LIN {X 0,Y 312.569,Z 218.829,A -85,B 0,C 180,E1 -15730.204,E2 -15730.204} C_VEL
LIN {X 0,Y 313.589,Z 221.679,A -85,B 0,C 180,E1 -15730.474,E2 -15730.474} C_VEL
LIN {X 0,Y 315.633,Z 224.126,A -85,B 0,C 180,E1 -15730.891,E2 -15730.891} C_VEL
LIN {X 0,Y 317.945,Z 227.629,A -85,B 0,C 180,E1 -15731.376,E2 -15731.376} C_VEL
LIN {X 0,Y 330.449,Z 246.954,A -85,B 0,C 180,E1 -15733.852,E2 -15733.852} C_VEL
LIN {X 0,Y 339.221,Z 262.018,A -85,B 0,C 180,E1 -15735.489,E2 -15735.489} C_VEL
LIN {X 0,Y 346.478,Z 276.506,A -85,B 0,C 180,E1 -15736.814,E2 -15736.814} C_VEL
LIN {X 0,Y 346.92,Z 277.621,A -85,B 0,C 180,E1 -15736.899,E2 -15736.899} C_VEL
LIN {X 0,Y 340.996,Z 419.211,A -85,B 0,C 180,E1 -15739.948,E2 -15739.948} C_VEL
LIN {X 0,Y 339.631,Z 436.329,A -85,B 0,C 180,E1 -15740.546,E2 -15740.546} C_VEL
LIN {X 0,Y 337.855,Z 452.225,A -85,B 0,C 180,E1 -15741.326,E2 -15741.326} C_VEL
LIN {X 0,Y 335.809,Z 467.786,A -85,B 0,C 180,E1 -15742.333,E2 -15742.333} C_VEL
LIN {X 0,Y 333.545,Z 482.265,A -85,B 0,C 180,E1 -15743.497,E2 -15743.497} C_VEL
LIN {X 0,Y 330.733,Z 497.251,A -85,B 0,C 180,E1 -15744.968,E2 -15744.968} C_VEL
LIN {X 0,Y 327.878,Z 510.986,A -85,B 0,C 180,E1 -15746.62,E2 -15746.62} C_VEL
LIN {X 0,Y 325.104,Z 523.666,A -85,B 0,C 180,E1 -15748.451,E2 -15748.451} C_VEL
LIN {X 0,Y 322.131,Z 536.293,A -85,B 0,C 180,E1 -15750.625,E2 -15750.625} C_VEL
LIN {X 0,Y 319.543,Z 547.053,A -85,B 0,C 180,E1 -15752.836,E2 -15752.836} C_VEL
LIN {X 0,Y 317.025,Z 557.47,A -85,B 0,C 180,E1 -15755.406,E2 -15755.406} C_VEL
LIN {X 0,Y 315.045,Z 566.149,A -85,B 0,C 180,E1 -15758.014,E2 -15758.014} C_VEL
LIN {X 0,Y 313.603,Z 572.562,A -85,B 0,C 180,E1 -15760.328,E2 -15760.328} C_VEL
LIN {X 0,Y 312.378,Z 578.726,A -85,B 0,C 180,E1 -15763.001,E2 -15763.001} C_VEL
LIN {X 0,Y 311.524,Z 583.601,A -85,B 0,C 180,E1 -15765.707,E2 -15765.707} C_VEL
LIN {X 0,Y 310.896,Z 587.382,A -85,B 0,C 180,E1 -15768.449,E2 -15768.449} C_VEL
LIN {X 0,Y 310.55,Z 590.089,A -85,B 0,C 180,E1 -15771.228,E2 -15771.228} C_VEL
LIN {X 0,Y 310.352,Z 591.614,A -85,B 0,C 180,E1 -15774.054,E2 -15774.054} C_VEL
LIN {X 0,Y 310.334,Z 592.053,A -85,B 0,C 180,E1 -15776.931,E2 -15776.931} C_VEL
LIN {X 0,Y 310.51,Z 591.326,A -85,B 0,C 180,E1 -15779.863,E2 -15779.863} C_VEL
LIN {X 0,Y 310.927,Z 588.932,A -85,B 0,C 180,E1 -15783.246,E2 -15783.246} C_VEL
LIN {X 0,Y 311.753,Z 584.791,A -85,B 0,C 180,E1 -15786.683,E2 -15786.683} C_VEL
LIN {X 0,Y 312.79,Z 579.753,A -85,B 0,C 180,E1 -15789.629,E2 -15789.629} C_VEL
LIN {X 0,Y 314.219,Z 573.616,A -85,B 0,C 180,E1 -15792.431,E2 -15792.431} C_VEL
LIN {X 0,Y 315.326,Z 569.216,A -85,B 0,C 180,E1 -15794.117,E2 -15794.117} C_VEL
LIN {X 0,Y 315.393,Z 566.63,A -85,B 0,C 180,E1 -15795.081,E2 -15795.081} C_VEL
LIN {X 0,Y 312.533,Z 557.734,A -85,B 0,C 180,E1 -15798.272,E2 -15798.272} C_VEL
LIN {X 0,Y 312.862,Z 554.516,A -85,B 0,C 180,E1 -15799.184,E2 -15799.184} C_VEL
LIN {X 0,Y 315.976,Z 543.99,A -85,B 0,C 180,E1 -15801.682,E2 -15801.682} C_VEL
LIN {X 0,Y 319.14,Z 533.152,A -85,B 0,C 180,E1 -15803.831,E2 -15803.831} C_VEL
LIN {X 0,Y 322.204,Z 521.844,A -85,B 0,C 180,E1 -15805.734,E2 -15805.734} C_VEL
LIN {X 0,Y 325.653,Z 508.462,A -85,B 0,C 180,E1 -15807.602,E2 -15807.602} C_VEL
LIN {X 0,Y 328.772,Z 495.26,A -85,B 0,C 180,E1 -15809.134,E2 -15809.134} C_VEL
LIN {X 0,Y 331.674,Z 481.349,A -85,B 0,C 180,E1 -15810.484,E2 -15810.484} C_VEL
LIN {X 0,Y 334.505,Z 465.783,A -85,B 0,C 180,E1 -15811.703,E2 -15811.703} C_VEL
LIN {X 0,Y 336.821,Z 449.961,A -85,B 0,C 180,E1 -15812.675,E2 -15812.675} C_VEL
LIN {X 0,Y 338.694,Z 433.873,A -85,B 0,C 180,E1 -15813.419,E2 -15813.419} C_VEL
LIN {X 0,Y 340.182,Z 416.337,A -85,B 0,C 180,E1 -15813.973,E2 -15813.973} C_VEL
LIN {X 0,Y 346.65,Z 282.972,A -85,B 0,C 180,E1 -15816.935,E2 -15816.935} C_VEL
LIN {X 0,Y 340.142,Z 270.114,A -85,B 0,C 180,E1 -15818.442,E2 -15818.442} C_VEL
LIN {X 0,Y 335.198,Z 261.466,A -85,B 0,C 180,E1 -15819.629,E2 -15819.629} C_VEL
LIN {X 0,Y 328.703,Z 251.5,A -85,B 0,C 180,E1 -15821.263,E2 -15821.263} C_VEL
LIN {X 0,Y 322.882,Z 243.203,A -85,B 0,C 180,E1 -15822.83,E2 -15822.83} C_VEL
LIN {X 0,Y 319.655,Z 238.87,A -85,B 0,C 180,E1 -15823.746,E2 -15823.746} C_VEL
LIN {X 0,Y 316.6,Z 234.714,A -85,B 0,C 180,E1 -15824.664,E2 -15824.664} C_VEL
LIN {X 0,Y 313.996,Z 231.244,A -85,B 0,C 180,E1 -15825.477,E2 -15825.477} C_VEL
LIN {X 0,Y 313.147,Z 230.084,A -85,B 0,C 180,E1 -15825.753,E2 -15825.753} C_VEL
LIN {X 0,Y 310.657,Z 227.254,A -85,B 0,C 180,E1 -15826.559,E2 -15826.559} C_VEL
LIN {X 0,Y 309.552,Z 225.243,A -85,B 0,C 180,E1 -15826.961,E2 -15826.961} C_VEL
LIN {X 0,Y 307.098,Z 223.278,A -85,B 0,C 180,E1 -15827.779,E2 -15827.779} C_VEL
LIN {X 0,Y 305.86,Z 220.899,A -85,B 0,C 180,E1 -15828.275,E2 -15828.275} C_VEL
LIN {X 0,Y 305.62,Z 219.711,A -85,B 0,C 180,E1 -15828.434,E2 -15828.434} C_VEL
LIN {X 0,Y 305.766,Z 219.711,A -85,B 0,C 180,E1 -15832.073,E2 -15832.073} C_VEL
LIN {X 0,Y 305.676,Z 219.722,A -85,B 0,C 180,E1 -15834.723,E2 -15834.723} C_VEL
LIN {X 0,Y 305.951,Z 219.685,A -85,B 0,C 180,E1 -15838.684,E2 -15838.684} C_VEL
LIN {X 0,Y 305.951,Z 219.686,A -85,B 0,C 180,E1 -15841.316,E2 -15841.316} C_VEL
LIN {X 0,Y 305.837,Z 219.7,A -85,B 0,C 180,E1 -15846.598,E2 -15846.598} C_VEL
LIN {X 0,Y 305.698,Z 219.717,A -85,B 0,C 180,E1 -15849.261,E2 -15849.261} C_VEL
LIN {X 0,Y 305.583,Z 219.729,A -85,B 0,C 180,E1 -15853.296,E2 -15853.296} C_VEL
LIN {X 0,Y 305.588,Z 219.727,A -85,B 0,C 180,E1 -15856.02,E2 -15856.02} C_VEL
LIN {X 0,Y 305.571,Z 219.729,A -85,B 0,C 180,E1 -15859.445,E2 -15859.445} C_VEL
LIN {X 0,Y 305.486,Z 219.746,A -85,B 0,C 180,E1 -15863.042,E2 -15863.042} C_VEL
LIN {X 0,Y 305.526,Z 219.736,A -85,B 0,C 180,E1 -15866.221,E2 -15866.221} C_VEL
LIN {X 0,Y 305.483,Z 219.742,A -85,B 0,C 180,E1 -15869.047,E2 -15869.047} C_VEL
LIN {X 0,Y 305.437,Z 219.751,A -85,B 0,C 180,E1 -15871.953,E2 -15871.953} C_VEL
LIN {X 0,Y 305.514,Z 219.86,A -85,B 0,C 180,E1 -15876.018,E2 -15876.018} C_VEL
LIN {X 0,Y 305.951,Z 221.601,A -85,B 0,C 180,E1 -15876.673,E2 -15876.673} C_VEL
LIN {X 0,Y 307.613,Z 224.865,A -85,B 0,C 180,E1 -15878.087,E2 -15878.087} C_VEL
LIN {X 0,Y 314.06,Z 233.766,A -85,B 0,C 180,E1 -15880.282,E2 -15880.282} C_VEL
LIN {X 0,Y 317.349,Z 238.402,A -85,B 0,C 180,E1 -15881.308,E2 -15881.308} C_VEL
LIN {X 0,Y 323.89,Z 248.152,A -85,B 0,C 180,E1 -15883.218,E2 -15883.218} C_VEL
LIN {X 0,Y 330.61,Z 259.152,A -85,B 0,C 180,E1 -15885.03,E2 -15885.03} C_VEL
LIN {X 0,Y 337.16,Z 270.828,A -85,B 0,C 180,E1 -15886.682,E2 -15886.682} C_VEL
LIN {X 0,Y 344.759,Z 286.276,A -85,B 0,C 180,E1 -15888.492,E2 -15888.492} C_VEL
LIN {X 0,Y 346.397,Z 289.941,A -85,B 0,C 180,E1 -15888.87,E2 -15888.87} C_VEL
LIN {X 0,Y 342.866,Z 363.369,A -85,B 0,C 180,E1 -15890.493,E2 -15890.493} C_VEL
LIN {X 0,Y 339.405,Z 435.134,A -85,B 0,C 180,E1 -15892.117,E2 -15892.117} C_VEL
LIN {X 0,Y 337.581,Z 452.624,A -85,B 0,C 180,E1 -15892.709,E2 -15892.709} C_VEL
LIN {X 0,Y 335.323,Z 469.014,A -85,B 0,C 180,E1 -15893.509,E2 -15893.509} C_VEL
LIN {X 0,Y 332.78,Z 484.339,A -85,B 0,C 180,E1 -15894.496,E2 -15894.496} C_VEL
LIN {X 0,Y 329.551,Z 500.237,A -85,B 0,C 180,E1 -15895.774,E2 -15895.774} C_VEL
LIN {X 0,Y 326.409,Z 514.583,A -85,B 0,C 180,E1 -15897.22,E2 -15897.22} C_VEL
LIN {X 0,Y 323.002,Z 528.277,A -85,B 0,C 180,E1 -15898.886,E2 -15898.886} C_VEL
LIN {X 0,Y 319.679,Z 540.731,A -85,B 0,C 180,E1 -15900.716,E2 -15900.716} C_VEL
LIN {X 0,Y 316.341,Z 552.857,A -85,B 0,C 180,E1 -15902.839,E2 -15902.839} C_VEL
LIN {X 0,Y 313.259,Z 563.818,A -85,B 0,C 180,E1 -15905.125,E2 -15905.125} C_VEL
LIN {X 0,Y 310.401,Z 574.161,A -85,B 0,C 180,E1 -15907.714,E2 -15907.714} C_VEL
LIN {X 0,Y 308.171,Z 582.797,A -85,B 0,C 180,E1 -15910.344,E2 -15910.344} C_VEL
LIN {X 0,Y 306.182,Z 590.845,A -85,B 0,C 180,E1 -15913.327,E2 -15913.327} C_VEL
LIN {X 0,Y 304.989,Z 596.69,A -85,B 0,C 180,E1 -15915.999,E2 -15915.999} C_VEL
LIN {X 0,Y 304.163,Z 601.391,A -85,B 0,C 180,E1 -15918.674,E2 -15918.674} C_VEL
LIN {X 0,Y 303.817,Z 604.222,A -85,B 0,C 180,E1 -15920.682,E2 -15920.682} C_VEL
LIN {X 0,Y 303.618,Z 607.009,A -85,B 0,C 180,E1 -15923.354,E2 -15923.354} C_VEL
LIN {X 0,Y 303.566,Z 608.885,A -85,B 0,C 180,E1 -15926.018,E2 -15926.018} C_VEL
LIN {X 0,Y 303.575,Z 609.682,A -85,B 0,C 180,E1 -15928.674,E2 -15928.674} C_VEL
LIN {X 0,Y 303.575,Z 609.59,A -85,B 0,C 180,E1 -15931.327,E2 -15931.327} C_VEL
LIN {X 0,Y 303.599,Z 608.416,A -85,B 0,C 180,E1 -15933.983,E2 -15933.983} C_VEL
LIN {X 0,Y 303.618,Z 606.325,A -85,B 0,C 180,E1 -15936.646,E2 -15936.646} C_VEL
LIN {X 0,Y 303.808,Z 603.111,A -85,B 0,C 180,E1 -15939.319,E2 -15939.319} C_VEL
LIN {X 0,Y 304.305,Z 598.874,A -85,B 0,C 180,E1 -15941.997,E2 -15941.997} C_VEL
LIN {X 0,Y 305.262,Z 593.244,A -85,B 0,C 180,E1 -15944.77,E2 -15944.77} C_VEL
LIN {X 0,Y 306.403,Z 586.766,A -85,B 0,C 180,E1 -15947.349,E2 -15947.349} C_VEL
LIN {X 0,Y 308.156,Z 578.729,A -85,B 0,C 180,E1 -15950.005,E2 -15950.005} C_VEL
LIN {X 0,Y 310.396,Z 569.109,A -85,B 0,C 180,E1 -15952.639,E2 -15952.639} C_VEL
LIN {X 0,Y 313.287,Z 557.586,A -85,B 0,C 180,E1 -15955.229,E2 -15955.229} C_VEL
LIN {X 0,Y 315.771,Z 547.009,A -85,B 0,C 180,E1 -15957.22,E2 -15957.22} C_VEL
LIN {X 0,Y 318.71,Z 534.598,A -85,B 0,C 180,E1 -15959.202,E2 -15959.202} C_VEL
LIN {X 0,Y 321.65,Z 521.958,A -85,B 0,C 180,E1 -15960.895,E2 -15960.895} C_VEL
LIN {X 0,Y 324.777,Z 507.198,A -85,B 0,C 180,E1 -15962.525,E2 -15962.525} C_VEL
LIN {X 0,Y 327.701,Z 491.892,A -85,B 0,C 180,E1 -15963.89,E2 -15963.89} C_VEL
LIN {X 0,Y 330.138,Z 476.607,A -85,B 0,C 180,E1 -15964.991,E2 -15964.991} C_VEL
LIN {X 0,Y 332.302,Z 459.741,A -85,B 0,C 180,E1 -15965.937,E2 -15965.937} C_VEL
LIN {X 0,Y 334.07,Z 443.602,A -85,B 0,C 180,E1 -15966.582,E2 -15966.582} C_VEL
LIN {X 0,Y 335.225,Z 427.63,A -85,B 0,C 180,E1 -15967.018,E2 -15967.018} C_VEL
LIN {X 0,Y 340.97,Z 287.709,A -85,B 0,C 180,E1 -15970.075,E2 -15970.075} C_VEL
LIN {X 0,Y 333.834,Z 272.618,A -85,B 0,C 180,E1 -15971.436,E2 -15971.436} C_VEL
LIN {X 0,Y 324.567,Z 254.726,A -85,B 0,C 180,E1 -15973.279,E2 -15973.279} C_VEL
LIN {X 0,Y 314.082,Z 236.733,A -85,B 0,C 180,E1 -15975.47,E2 -15975.47} C_VEL
LIN {X 0,Y 308.14,Z 226.968,A -85,B 0,C 180,E1 -15976.825,E2 -15976.825} C_VEL
LIN {X 0,Y 305.419,Z 219.741,A -85,B 0,C 180,E1 -15978.827,E2 -15978.827} C_VEL
LIN {X 0,Y 305.46,Z 219.751,A -85,B 0,C 180,E1 -15981.595,E2 -15981.595} C_VEL
LIN {X 0,Y 305.46,Z 219.738,A -85,B 0,C 180,E1 -15984.887,E2 -15984.887} C_VEL
LIN {X 0,Y 305.447,Z 219.727,A -85,B 0,C 180,E1 -15988.356,E2 -15988.356} C_VEL
LIN {X 0,Y 305.512,Z 219.744,A -85,B 0,C 180,E1 -15991.113,E2 -15991.113} C_VEL
LIN {X 0,Y 305.563,Z 219.708,A -85,B 0,C 180,E1 -15994.087,E2 -15994.087} C_VEL
LIN {X 0,Y 305.493,Z 219.737,A -85,B 0,C 180,E1 -15998.402,E2 -15998.402} C_VEL
LIN {X 0,Y 305.541,Z 219.706,A -85,B 0,C 180,E1 -16001.215,E2 -16001.215} C_VEL
LIN {X 0,Y 305.624,Z 219.724,A -85,B 0,C 180,E1 -16005.348,E2 -16005.348} C_VEL
LIN {X 0,Y 305.622,Z 219.693,A -85,B 0,C 180,E1 -16009.399,E2 -16009.399} C_VEL
LIN {X 0,Y 305.769,Z 219.708,A -85,B 0,C 180,E1 -16012.073,E2 -16012.073} C_VEL
LIN {X 0,Y 305.679,Z 219.702,A -85,B 0,C 180,E1 -16014.723,E2 -16014.723} C_VEL
LIN {X 0,Y 305.953,Z 219.652,A -85,B 0,C 180,E1 -16018.684,E2 -16018.684} C_VEL
LIN {X 0,Y 305.955,Z 219.685,A -85,B 0,C 180,E1 -16021.316,E2 -16021.316} C_VEL
LIN {X 0,Y 305.84,Z 219.686,A -85,B 0,C 180,E1 -16026.601,E2 -16026.601} C_VEL
LIN {X 0,Y 305.702,Z 219.715,A -85,B 0,C 180,E1 -16029.261,E2 -16029.261} C_VEL
LIN {X 0,Y 305.586,Z 219.717,A -85,B 0,C 180,E1 -16033.296,E2 -16033.296} C_VEL
LIN {X 0,Y 305.592,Z 219.728,A -85,B 0,C 180,E1 -16036.02,E2 -16036.02} C_VEL
LIN {X 0,Y 305.575,Z 219.709,A -85,B 0,C 180,E1 -16039.445,E2 -16039.445} C_VEL
LIN {X 0,Y 305.489,Z 219.742,A -85,B 0,C 180,E1 -16043.041,E2 -16043.041} C_VEL
LIN {X 0,Y 305.553,Z 219.715,A -85,B 0,C 180,E1 -16046.23,E2 -16046.23} C_VEL
LIN {X 0,Y 305.502,Z 219.743,A -85,B 0,C 180,E1 -16049.052,E2 -16049.052} C_VEL
LIN {X 0,Y 305.464,Z 219.736,A -85,B 0,C 180,E1 -16053.517,E2 -16053.517} C_VEL
LIN {X 0,Y 305.471,Z 219.738,A -85,B 0,C 180,E1 -16056.74,E2 -16056.74} C_VEL
LIN {X 0,Y 305.454,Z 219.748,A -85,B 0,C 180,E1 -16060.6,E2 -16060.6} C_VEL
LIN {X 0,Y 305.424,Z 219.735,A -85,B 0,C 180,E1 -16063.655,E2 -16063.655} C_VEL
LIN {X 0,Y 305.454,Z 219.744,A -85,B 0,C 180,E1 -16067.414,E2 -16067.414} C_VEL
LIN {X 0,Y 305.475,Z 219.747,A -85,B 0,C 180,E1 -16071.598,E2 -16071.598} C_VEL
LIN {X 0,Y 305.461,Z 219.736,A -85,B 0,C 180,E1 -16074.887,E2 -16074.887} C_VEL
LIN {X 0,Y 305.451,Z 219.735,A -85,B 0,C 180,E1 -16078.355,E2 -16078.355} C_VEL
LIN {X 0,Y 305.52,Z 219.742,A -85,B 0,C 180,E1 -16081.114,E2 -16081.114} C_VEL
LIN {X 0,Y 305.571,Z 219.732,A -85,B 0,C 180,E1 -16084.088,E2 -16084.088} C_VEL
LIN {X 0,Y 305.511,Z 219.733,A -85,B 0,C 180,E1 -16088.722,E2 -16088.722} C_VEL
LIN {X 0,Y 305.526,Z 219.862,A -85,B 0,C 180,E1 -16089.021,E2 -16089.021} C_VEL
LIN {X 0,Y 306.552,Z 222.628,A -85,B 0,C 180,E1 -16089.295,E2 -16089.295} C_VEL
LIN {X 0,Y 308.681,Z 225.163,A -85,B 0,C 180,E1 -16089.75,E2 -16089.75} C_VEL
LIN {X 0,Y 310.838,Z 228.393,A -85,B 0,C 180,E1 -16090.225,E2 -16090.225} C_VEL
LIN {X 0,Y 321.959,Z 245.231,A -85,B 0,C 180,E1 -16092.545,E2 -16092.545} C_VEL
LIN {X 0,Y 330.594,Z 259.454,A -85,B 0,C 180,E1 -16094.234,E2 -16094.234} C_VEL
LIN {X 0,Y 336.365,Z 269.967,A -85,B 0,C 180,E1 -16095.329,E2 -16095.329} C_VEL
LIN {X 0,Y 341.118,Z 279.595,A -85,B 0,C 180,E1 -16096.219,E2 -16096.219} C_VEL
LIN {X 0,Y 335.132,Z 419.139,A -85,B 0,C 180,E1 -16099.274,E2 -16099.274} C_VEL
LIN {X 0,Y 333.716,Z 436.368,A -85,B 0,C 180,E1 -16099.879,E2 -16099.879} C_VEL
LIN {X 0,Y 331.815,Z 452.948,A -85,B 0,C 180,E1 -16100.706,E2 -16100.706} C_VEL
LIN {X 0,Y 329.677,Z 468.427,A -85,B 0,C 180,E1 -16101.726,E2 -16101.726} C_VEL
LIN {X 0,Y 327.361,Z 482.815,A -85,B 0,C 180,E1 -16102.909,E2 -16102.909} C_VEL
LIN {X 0,Y 324.448,Z 497.796,A -85,B 0,C 180,E1 -16104.405,E2 -16104.405} C_VEL
LIN {X 0,Y 321.504,Z 511.467,A -85,B 0,C 180,E1 -16106.083,E2 -16106.083} C_VEL
LIN {X 0,Y 318.822,Z 523.141,A -85,B 0,C 180,E1 -16107.789,E2 -16107.789} C_VEL
LIN {X 0,Y 315.998,Z 534.828,A -85,B 0,C 180,E1 -16109.795,E2 -16109.795} C_VEL
LIN {X 0,Y 313.384,Z 545.28,A -85,B 0,C 180,E1 -16111.927,E2 -16111.927} C_VEL
LIN {X 0,Y 310.805,Z 555.383,A -85,B 0,C 180,E1 -16114.383,E2 -16114.383} C_VEL
LIN {X 0,Y 308.713,Z 563.923,A -85,B 0,C 180,E1 -16116.864,E2 -16116.864} C_VEL
LIN {X 0,Y 307.114,Z 570.736,A -85,B 0,C 180,E1 -16119.217,E2 -16119.217} C_VEL
LIN {X 0,Y 305.74,Z 577.196,A -85,B 0,C 180,E1 -16121.939,E2 -16121.939} C_VEL
LIN {X 0,Y 304.708,Z 582.483,A -85,B 0,C 180,E1 -16124.697,E2 -16124.697} C_VEL
LIN {X 0,Y 303.991,Z 586.603,A -85,B 0,C 180,E1 -16127.49,E2 -16127.49} C_VEL
LIN {X 0,Y 303.515,Z 589.576,A -85,B 0,C 180,E1 -16130.323,E2 -16130.323} C_VEL
LIN {X 0,Y 303.271,Z 591.502,A -85,B 0,C 180,E1 -16133.2,E2 -16133.2} C_VEL
LIN {X 0,Y 303.219,Z 592.26,A -85,B 0,C 180,E1 -16136.127,E2 -16136.127} C_VEL
LIN {X 0,Y 303.36,Z 591.84,A -85,B 0,C 180,E1 -16139.111,E2 -16139.111} C_VEL
LIN {X 0,Y 303.642,Z 590.209,A -85,B 0,C 180,E1 -16142.163,E2 -16142.163} C_VEL
LIN {X 0,Y 304.273,Z 587.239,A -85,B 0,C 180,E1 -16145.27,E2 -16145.27} C_VEL
LIN {X 0,Y 305.238,Z 582.667,A -85,B 0,C 180,E1 -16148.479,E2 -16148.479} C_VEL
LIN {X 0,Y 306.689,Z 576.602,A -85,B 0,C 180,E1 -16151.647,E2 -16151.647} C_VEL
LIN {X 0,Y 308.505,Z 569.741,A -85,B 0,C 180,E1 -16154.467,E2 -16154.467} C_VEL
LIN {X 0,Y 310.901,Z 561.24,A -85,B 0,C 180,E1 -16157.3,E2 -16157.3} C_VEL
LIN {X 0,Y 312.862,Z 554.516,A -85,B 0,C 180,E1 -16159.184,E2 -16159.184} C_VEL
LIN {X 0,Y 313.25,Z 551.252,A -85,B 0,C 180,E1 -16160.082,E2 -16160.082} C_VEL
LIN {X 0,Y 311.457,Z 540.284,A -85,B 0,C 180,E1 -16163.088,E2 -16163.088} C_VEL
LIN {X 0,Y 312.049,Z 536.454,A -85,B 0,C 180,E1 -16163.913,E2 -16163.913} C_VEL
LIN {X 0,Y 315.472,Z 524.42,A -85,B 0,C 180,E1 -16166.05,E2 -16166.05} C_VEL
LIN {X 0,Y 319.091,Z 511.357,A -85,B 0,C 180,E1 -16167.966,E2 -16167.966} C_VEL
LIN {X 0,Y 322.175,Z 498.973,A -85,B 0,C 180,E1 -16169.502,E2 -16169.502} C_VEL
LIN {X 0,Y 325.456,Z 484.325,A -85,B 0,C 180,E1 -16170.992,E2 -16170.992} C_VEL
LIN {X 0,Y 328.363,Z 469.451,A -85,B 0,C 180,E1 -16172.218,E2 -16172.218} C_VEL
LIN {X 0,Y 330.743,Z 454.966,A -85,B 0,C 180,E1 -16173.182,E2 -16173.182} C_VEL
LIN {X 0,Y 332.751,Z 439.646,A -85,B 0,C 180,E1 -16173.983,E2 -16173.983} C_VEL
LIN {X 0,Y 334.379,Z 423.357,A -85,B 0,C 180,E1 -16174.582,E2 -16174.582} C_VEL
LIN {X 0,Y 335.785,Z 398.674,A -85,B 0,C 180,E1 -16175.187,E2 -16175.187} C_VEL
LIN {X 0,Y 341.519,Z 285.669,A -85,B 0,C 180,E1 -16177.71,E2 -16177.71} C_VEL
LIN {X 0,Y 335.762,Z 274.293,A -85,B 0,C 180,E1 -16179.098,E2 -16179.098} C_VEL
LIN {X 0,Y 331.39,Z 266.453,A -85,B 0,C 180,E1 -16180.198,E2 -16180.198} C_VEL
LIN {X 0,Y 324.525,Z 255.848,A -85,B 0,C 180,E1 -16181.992,E2 -16181.992} C_VEL
LIN {X 0,Y 319.039,Z 248.008,A -85,B 0,C 180,E1 -16183.535,E2 -16183.535} C_VEL
LIN {X 0,Y 316.21,Z 244.147,A -85,B 0,C 180,E1 -16184.377,E2 -16184.377} C_VEL
LIN {X 0,Y 313.482,Z 240.367,A -85,B 0,C 180,E1 -16185.228,E2 -16185.228} C_VEL
LIN {X 0,Y 310.182,Z 235.952,A -85,B 0,C 180,E1 -16186.307,E2 -16186.307} C_VEL
LIN {X 0,Y 307.54,Z 232.58,A -85,B 0,C 180,E1 -16187.21,E2 -16187.21} C_VEL
LIN {X 0,Y 306.712,Z 231.384,A -85,B 0,C 180,E1 -16187.511,E2 -16187.511} C_VEL
LIN {X 0,Y 304.265,Z 228.977,A -85,B 0,C 180,E1 -16188.382,E2 -16188.382} C_VEL
LIN {X 0,Y 302.648,Z 226.153,A -85,B 0,C 180,E1 -16189.04,E2 -16189.04} C_VEL
LIN {X 0,Y 300.243,Z 224.347,A -85,B 0,C 180,E1 -16189.932,E2 -16189.932} C_VEL
LIN {X 0,Y 298.977,Z 222.103,A -85,B 0,C 180,E1 -16190.486,E2 -16190.486} C_VEL
LIN {X 0,Y 298.669,Z 220.592,A -85,B 0,C 180,E1 -16190.729,E2 -16190.729} C_VEL
LIN {X 0,Y 298.769,Z 220.577,A -85,B 0,C 180,E1 -16193.245,E2 -16193.245} C_VEL
LIN {X 0,Y 298.918,Z 220.56,A -85,B 0,C 180,E1 -16198.653,E2 -16198.653} C_VEL
LIN {X 0,Y 298.918,Z 220.562,A -85,B 0,C 180,E1 -16201.347,E2 -16201.347} C_VEL
LIN {X 0,Y 298.782,Z 220.58,A -85,B 0,C 180,E1 -16206.754,E2 -16206.754} C_VEL
LIN {X 0,Y 298.63,Z 220.599,A -85,B 0,C 180,E1 -16209.482,E2 -16209.482} C_VEL
LIN {X 0,Y 298.547,Z 220.604,A -85,B 0,C 180,E1 -16213.616,E2 -16213.616} C_VEL
LIN {X 0,Y 298.543,Z 220.604,A -85,B 0,C 180,E1 -16216.409,E2 -16216.409} C_VEL
LIN {X 0,Y 298.506,Z 220.61,A -85,B 0,C 180,E1 -16219.655,E2 -16219.655} C_VEL
LIN {X 0,Y 298.453,Z 220.618,A -85,B 0,C 180,E1 -16223.598,E2 -16223.598} C_VEL
LIN {X 0,Y 298.482,Z 220.613,A -85,B 0,C 180,E1 -16226.575,E2 -16226.575} C_VEL
LIN {X 0,Y 298.411,Z 220.624,A -85,B 0,C 180,E1 -16229.642,E2 -16229.642} C_VEL
LIN {X 0,Y 298.426,Z 220.685,A -85,B 0,C 180,E1 -16233.907,E2 -16233.907} C_VEL
LIN {X 0,Y 299.354,Z 223.361,A -85,B 0,C 180,E1 -16235.112,E2 -16235.112} C_VEL
LIN {X 0,Y 300.441,Z 224.75,A -85,B 0,C 180,E1 -16235.789,E2 -16235.789} C_VEL
LIN {X 0,Y 302.599,Z 228.072,A -85,B 0,C 180,E1 -16236.674,E2 -16236.674} C_VEL
LIN {X 0,Y 305.308,Z 231.386,A -85,B 0,C 180,E1 -16237.694,E2 -16237.694} C_VEL
LIN {X 0,Y 311.192,Z 239.615,A -85,B 0,C 180,E1 -16239.766,E2 -16239.766} C_VEL
LIN {X 0,Y 314.353,Z 244.238,A -85,B 0,C 180,E1 -16240.795,E2 -16240.795} C_VEL
LIN {X 0,Y 320.383,Z 253.329,A -85,B 0,C 180,E1 -16242.62,E2 -16242.62} C_VEL
LIN {X 0,Y 327.747,Z 265.663,A -85,B 0,C 180,E1 -16244.677,E2 -16244.677} C_VEL
LIN {X 0,Y 333.797,Z 276.856,A -85,B 0,C 180,E1 -16246.256,E2 -16246.256} C_VEL
LIN {X 0,Y 340.947,Z 291.732,A -85,B 0,C 180,E1 -16248.018,E2 -16248.018} C_VEL
LIN {X 0,Y 341.275,Z 292.503,A -85,B 0,C 180,E1 -16248.099,E2 -16248.099} C_VEL
LIN {X 0,Y 335.393,Z 408.882,A -85,B 0,C 180,E1 -16250.69,E2 -16250.69} C_VEL
LIN {X 0,Y 333.935,Z 436.305,A -85,B 0,C 180,E1 -16251.357,E2 -16251.357} C_VEL
LIN {X 0,Y 332.089,Z 453.273,A -85,B 0,C 180,E1 -16251.948,E2 -16251.948} C_VEL
LIN {X 0,Y 329.69,Z 469.884,A -85,B 0,C 180,E1 -16252.782,E2 -16252.782} C_VEL
LIN {X 0,Y 327.044,Z 484.917,A -85,B 0,C 180,E1 -16253.776,E2 -16253.776} C_VEL
LIN {X 0,Y 323.728,Z 500.616,A -85,B 0,C 180,E1 -16255.07,E2 -16255.07} C_VEL
LIN {X 0,Y 320.429,Z 514.814,A -85,B 0,C 180,E1 -16256.523,E2 -16256.523} C_VEL
LIN {X 0,Y 316.9,Z 528.499,A -85,B 0,C 180,E1 -16258.217,E2 -16258.217} C_VEL
LIN {X 0,Y 313.457,Z 540.884,A -85,B 0,C 180,E1 -16260.076,E2 -16260.076} C_VEL
LIN {X 0,Y 310.184,Z 552.186,A -85,B 0,C 180,E1 -16262.084,E2 -16262.084} C_VEL
LIN {X 0,Y 307.16,Z 562.462,A -85,B 0,C 180,E1 -16264.233,E2 -16264.233} C_VEL
LIN {X 0,Y 304.089,Z 572.922,A -85,B 0,C 180,E1 -16266.866,E2 -16266.866} C_VEL
LIN {X 0,Y 301.634,Z 581.728,A -85,B 0,C 180,E1 -16269.544,E2 -16269.544} C_VEL
LIN {X 0,Y 299.67,Z 589.128,A -85,B 0,C 180,E1 -16272.25,E2 -16272.25} C_VEL
LIN {X 0,Y 298.232,Z 595.426,A -85,B 0,C 180,E1 -16275.057,E2 -16275.057} C_VEL
LIN {X 0,Y 297.327,Z 600.166,A -85,B 0,C 180,E1 -16277.718,E2 -16277.718} C_VEL
LIN {X 0,Y 296.736,Z 604.069,A -85,B 0,C 180,E1 -16280.457,E2 -16280.457} C_VEL
LIN {X 0,Y 296.533,Z 606.841,A -85,B 0,C 180,E1 -16283.195,E2 -16283.195} C_VEL
LIN {X 0,Y 296.468,Z 608.698,A -85,B 0,C 180,E1 -16285.922,E2 -16285.922} C_VEL
LIN {X 0,Y 296.493,Z 609.482,A -85,B 0,C 180,E1 -16288.642,E2 -16288.642} C_VEL
LIN {X 0,Y 296.494,Z 609.369,A -85,B 0,C 180,E1 -16291.359,E2 -16291.359} C_VEL
LIN {X 0,Y 296.496,Z 608.18,A -85,B 0,C 180,E1 -16294.078,E2 -16294.078} C_VEL
LIN {X 0,Y 296.533,Z 606.063,A -85,B 0,C 180,E1 -16296.806,E2 -16296.806} C_VEL
LIN {X 0,Y 296.821,Z 601.913,A -85,B 0,C 180,E1 -16300.229,E2 -16300.229} C_VEL
LIN {X 0,Y 297.726,Z 596.03,A -85,B 0,C 180,E1 -16303.654,E2 -16303.654} C_VEL
LIN {X 0,Y 298.784,Z 589.928,A -85,B 0,C 180,E1 -16306.396,E2 -16306.396} C_VEL
LIN {X 0,Y 300.449,Z 582.559,A -85,B 0,C 180,E1 -16309.116,E2 -16309.116} C_VEL
LIN {X 0,Y 302.462,Z 573.722,A -85,B 0,C 180,E1 -16311.825,E2 -16311.825} C_VEL
LIN {X 0,Y 305.175,Z 563.162,A -85,B 0,C 180,E1 -16314.49,E2 -16314.49} C_VEL
LIN {X 0,Y 308.037,Z 552.164,A -85,B 0,C 180,E1 -16316.783,E2 -16316.783} C_VEL
LIN {X 0,Y 310.688,Z 541.188,A -85,B 0,C 180,E1 -16318.731,E2 -16318.731} C_VEL
LIN {X 0,Y 313.813,Z 528.472,A -85,B 0,C 180,E1 -16320.63,E2 -16320.63} C_VEL
LIN {X 0,Y 316.972,Z 514.747,A -85,B 0,C 180,E1 -16322.333,E2 -16322.333} C_VEL
LIN {X 0,Y 320.081,Z 499.686,A -85,B 0,C 180,E1 -16323.859,E2 -16323.859} C_VEL
LIN {X 0,Y 322.75,Z 485.142,A -85,B 0,C 180,E1 -16325.052,E2 -16325.052} C_VEL
LIN {X 0,Y 325.135,Z 469.466,A -85,B 0,C 180,E1 -16326.088,E2 -16326.088} C_VEL
LIN {X 0,Y 327.11,Z 453.669,A -85,B 0,C 180,E1 -16326.887,E2 -16326.887} C_VEL
LIN {X 0,Y 328.85,Z 436.439,A -85,B 0,C 180,E1 -16327.482,E2 -16327.482} C_VEL
LIN {X 0,Y 330.945,Z 388.089,A -85,B 0,C 180,E1 -16328.595,E2 -16328.595} C_VEL
LIN {X 0,Y 335.289,Z 290.092,A -85,B 0,C 180,E1 -16330.748,E2 -16330.748} C_VEL
LIN {X 0,Y 328.655,Z 276,A -85,B 0,C 180,E1 -16332.062,E2 -16332.062} C_VEL
LIN {X 0,Y 320.133,Z 259.451,A -85,B 0,C 180,E1 -16333.804,E2 -16333.804} C_VEL
LIN {X 0,Y 310.032,Z 241.85,A -85,B 0,C 180,E1 -16335.978,E2 -16335.978} C_VEL
LIN {X 0,Y 300.653,Z 226.753,A -85,B 0,C 180,E1 -16338.17,E2 -16338.17} C_VEL
LIN {X 0,Y 298.404,Z 220.614,A -85,B 0,C 180,E1 -16339.965,E2 -16339.965} C_VEL
LIN {X 0,Y 298.403,Z 220.609,A -85,B 0,C 180,E1 -16343.928,E2 -16343.928} C_VEL
LIN {X 0,Y 298.393,Z 220.613,A -85,B 0,C 180,E1 -16347.2,E2 -16347.2} C_VEL
LIN {X 0,Y 298.426,Z 220.623,A -85,B 0,C 180,E1 -16350.616,E2 -16350.616} C_VEL
LIN {X 0,Y 298.475,Z 220.592,A -85,B 0,C 180,E1 -16353.477,E2 -16353.477} C_VEL
LIN {X 0,Y 298.434,Z 220.623,A -85,B 0,C 180,E1 -16356.697,E2 -16356.697} C_VEL
LIN {X 0,Y 298.503,Z 220.58,A -85,B 0,C 180,E1 -16360.754,E2 -16360.754} C_VEL
LIN {X 0,Y 298.584,Z 220.602,A -85,B 0,C 180,E1 -16364.994,E2 -16364.994} C_VEL
LIN {X 0,Y 298.581,Z 220.567,A -85,B 0,C 180,E1 -16369.146,E2 -16369.146} C_VEL
LIN {X 0,Y 298.715,Z 220.586,A -85,B 0,C 180,E1 -16371.885,E2 -16371.885} C_VEL
LIN {X 0,Y 298.65,Z 220.579,A -85,B 0,C 180,E1 -16374.599,E2 -16374.599} C_VEL
LIN {X 0,Y 298.92,Z 220.527,A -85,B 0,C 180,E1 -16378.653,E2 -16378.653} C_VEL
LIN {X 0,Y 298.921,Z 220.562,A -85,B 0,C 180,E1 -16381.347,E2 -16381.347} C_VEL
LIN {X 0,Y 298.786,Z 220.566,A -85,B 0,C 180,E1 -16386.754,E2 -16386.754} C_VEL
LIN {X 0,Y 298.634,Z 220.595,A -85,B 0,C 180,E1 -16389.482,E2 -16389.482} C_VEL
LIN {X 0,Y 298.55,Z 220.596,A -85,B 0,C 180,E1 -16393.615,E2 -16393.615} C_VEL
LIN {X 0,Y 298.547,Z 220.602,A -85,B 0,C 180,E1 -16396.409,E2 -16396.409} C_VEL
LIN {X 0,Y 298.51,Z 220.59,A -85,B 0,C 180,E1 -16399.654,E2 -16399.654} C_VEL
LIN {X 0,Y 298.456,Z 220.611,A -85,B 0,C 180,E1 -16403.598,E2 -16403.598} C_VEL
LIN {X 0,Y 298.491,Z 220.598,A -85,B 0,C 180,E1 -16406.574,E2 -16406.574} C_VEL
LIN {X 0,Y 298.423,Z 220.622,A -85,B 0,C 180,E1 -16409.641,E2 -16409.641} C_VEL
LIN {X 0,Y 298.395,Z 220.609,A -85,B 0,C 180,E1 -16412.8,E2 -16412.8} C_VEL
LIN {X 0,Y 298.443,Z 220.611,A -85,B 0,C 180,E1 -16416.807,E2 -16416.807} C_VEL
LIN {X 0,Y 298.386,Z 220.63,A -85,B 0,C 180,E1 -16421.088,E2 -16421.088} C_VEL
LIN {X 0,Y 298.398,Z 220.613,A -85,B 0,C 180,E1 -16423.103,E2 -16423.103} C_VEL
LIN {X 0,Y 298.402,Z 220.628,A -85,B 0,C 180,E1 -16426.921,E2 -16426.921} C_VEL
LIN {X 0,Y 298.403,Z 220.626,A -85,B 0,C 180,E1 -16431.006,E2 -16431.006} C_VEL
LIN {X 0,Y 298.417,Z 220.608,A -85,B 0,C 180,E1 -16433.93,E2 -16433.93} C_VEL
LIN {X 0,Y 298.394,Z 220.616,A -85,B 0,C 180,E1 -16437.983,E2 -16437.983} C_VEL
LIN {X 0,Y 298.463,Z 220.612,A -85,B 0,C 180,E1 -16441.904,E2 -16441.904} C_VEL
LIN {X 0,Y 298.485,Z 220.616,A -85,B 0,C 180,E1 -16444.924,E2 -16444.924} C_VEL
LIN {X 0,Y 298.462,Z 220.62,A -85,B 0,C 180,E1 -16447.722,E2 -16447.722} C_VEL
LIN {X 0,Y 299.551,Z 223.613,A -85,B 0,C 180,E1 -16448.059,E2 -16448.059} C_VEL
LIN {X 0,Y 301.577,Z 225.883,A -85,B 0,C 180,E1 -16448.513,E2 -16448.513} C_VEL
LIN {X 0,Y 303.634,Z 229.157,A -85,B 0,C 180,E1 -16448.997,E2 -16448.997} C_VEL
LIN {X 0,Y 305.355,Z 231.622,A -85,B 0,C 180,E1 -16449.385,E2 -16449.385} C_VEL
LIN {X 0,Y 308.773,Z 236.531,A -85,B 0,C 180,E1 -16450.14,E2 -16450.14} C_VEL
LIN {X 0,Y 320.148,Z 254.042,A -85,B 0,C 180,E1 -16452.536,E2 -16452.536} C_VEL
LIN {X 0,Y 329.846,Z 270.783,A -85,B 0,C 180,E1 -16454.455,E2 -16454.455} C_VEL
LIN {X 0,Y 335.387,Z 281.991,A -85,B 0,C 180,E1 -16455.535,E2 -16455.535} C_VEL
LIN {X 0,Y 329.28,Z 419.252,A -85,B 0,C 180,E1 -16458.582,E2 -16458.582} C_VEL
LIN {X 0,Y 327.846,Z 436.31,A -85,B 0,C 180,E1 -16459.189,E2 -16459.189} C_VEL
LIN {X 0,Y 325.966,Z 452.322,A -85,B 0,C 180,E1 -16459.989,E2 -16459.989} C_VEL
LIN {X 0,Y 323.593,Z 468.98,A -85,B 0,C 180,E1 -16461.098,E2 -16461.098} C_VEL
LIN {X 0,Y 320.835,Z 484.927,A -85,B 0,C 180,E1 -16462.447,E2 -16462.447} C_VEL
LIN {X 0,Y 318.068,Z 498.812,A -85,B 0,C 180,E1 -16463.886,E2 -16463.886} C_VEL
LIN {X 0,Y 314.861,Z 513.087,A -85,B 0,C 180,E1 -16465.679,E2 -16465.679} C_VEL
LIN {X 0,Y 312.115,Z 524.539,A -85,B 0,C 180,E1 -16467.418,E2 -16467.418} C_VEL
LIN {X 0,Y 309.047,Z 536.685,A -85,B 0,C 180,E1 -16469.592,E2 -16469.592} C_VEL
LIN {X 0,Y 306.163,Z 547.802,A -85,B 0,C 180,E1 -16471.973,E2 -16471.973} C_VEL
LIN {X 0,Y 303.465,Z 558.001,A -85,B 0,C 180,E1 -16474.599,E2 -16474.599} C_VEL
LIN {X 0,Y 301.263,Z 566.828,A -85,B 0,C 180,E1 -16477.371,E2 -16477.371} C_VEL
LIN {X 0,Y 299.446,Z 574.333,A -85,B 0,C 180,E1 -16480.268,E2 -16480.268} C_VEL
LIN {X 0,Y 298.214,Z 579.95,A -85,B 0,C 180,E1 -16482.937,E2 -16482.937} C_VEL
LIN {X 0,Y 297.303,Z 584.721,A -85,B 0,C 180,E1 -16485.774,E2 -16485.774} C_VEL
LIN {X 0,Y 296.678,Z 588.268,A -85,B 0,C 180,E1 -16488.638,E2 -16488.638} C_VEL
LIN {X 0,Y 296.367,Z 590.279,A -85,B 0,C 180,E1 -16490.836,E2 -16490.836} C_VEL
LIN {X 0,Y 296.164,Z 591.926,A -85,B 0,C 180,E1 -16493.791,E2 -16493.791} C_VEL
LIN {X 0,Y 296.141,Z 592.495,A -85,B 0,C 180,E1 -16496.801,E2 -16496.801} C_VEL
LIN {X 0,Y 296.302,Z 591.836,A -85,B 0,C 180,E1 -16499.873,E2 -16499.873} C_VEL
LIN {X 0,Y 296.676,Z 589.895,A -85,B 0,C 180,E1 -16503.013,E2 -16503.013} C_VEL
LIN {X 0,Y 297.453,Z 586.61,A -85,B 0,C 180,E1 -16506.204,E2 -16506.204} C_VEL
LIN {X 0,Y 298.563,Z 581.82,A -85,B 0,C 180,E1 -16509.461,E2 -16509.461} C_VEL
LIN {X 0,Y 299.805,Z 577.013,A -85,B 0,C 180,E1 -16511.975,E2 -16511.975} C_VEL
LIN {X 0,Y 301.86,Z 569.551,A -85,B 0,C 180,E1 -16515.108,E2 -16515.108} C_VEL
LIN {X 0,Y 304.427,Z 561.029,A -85,B 0,C 180,E1 -16517.972,E2 -16517.972} C_VEL
LIN {X 0,Y 307.202,Z 552.13,A -85,B 0,C 180,E1 -16520.448,E2 -16520.448} C_VEL
LIN {X 0,Y 310.517,Z 541.434,A -85,B 0,C 180,E1 -16522.921,E2 -16522.921} C_VEL
LIN {X 0,Y 312.049,Z 536.454,A -85,B 0,C 180,E1 -16523.913,E2 -16523.913} C_VEL
LIN {X 0,Y 312.663,Z 532.572,A -85,B 0,C 180,E1 -16524.723,E2 -16524.723} C_VEL
LIN {X 0,Y 311.479,Z 520.379,A -85,B 0,C 180,E1 -16527.352,E2 -16527.352} C_VEL
LIN {X 0,Y 311.852,Z 516.81,A -85,B 0,C 180,E1 -16527.97,E2 -16527.97} C_VEL
LIN {X 0,Y 312.227,Z 515.316,A -85,B 0,C 180,E1 -16528.195,E2 -16528.195} C_VEL
LIN {X 0,Y 315.783,Z 501.826,A -85,B 0,C 180,E1 -16529.956,E2 -16529.956} C_VEL
LIN {X 0,Y 319.233,Z 487.439,A -85,B 0,C 180,E1 -16531.499,E2 -16531.499} C_VEL
LIN {X 0,Y 322.229,Z 473.294,A -85,B 0,C 180,E1 -16532.741,E2 -16532.741} C_VEL
LIN {X 0,Y 324.948,Z 457.807,A -85,B 0,C 180,E1 -16533.838,E2 -16533.838} C_VEL
LIN {X 0,Y 327.126,Z 442.167,A -85,B 0,C 180,E1 -16534.688,E2 -16534.688} C_VEL
LIN {X 0,Y 328.938,Z 425.833,A -85,B 0,C 180,E1 -16535.325,E2 -16535.325} C_VEL
LIN {X 0,Y 330.309,Z 404.581,A -85,B 0,C 180,E1 -16535.885,E2 -16535.885} C_VEL
LIN {X 0,Y 336.447,Z 288.344,A -85,B 0,C 180,E1 -16538.517,E2 -16538.517} C_VEL
LIN {X 0,Y 329.625,Z 274.85,A -85,B 0,C 180,E1 -16540.258,E2 -16540.258} C_VEL
LIN {X 0,Y 323.364,Z 264.693,A -85,B 0,C 180,E1 -16541.918,E2 -16541.918} C_VEL
LIN {X 0,Y 316.749,Z 254.78,A -85,B 0,C 180,E1 -16543.815,E2 -16543.815} C_VEL
LIN {X 0,Y 310.638,Z 246.27,A -85,B 0,C 180,E1 -16545.731,E2 -16545.731} C_VEL
LIN {X 0,Y 307.335,Z 241.868,A -85,B 0,C 180,E1 -16546.844,E2 -16546.844} C_VEL
LIN {X 0,Y 304.599,Z 238.089,A -85,B 0,C 180,E1 -16547.835,E2 -16547.835} C_VEL
LIN {X 0,Y 301.448,Z 234.6,A -85,B 0,C 180,E1 -16549.006,E2 -16549.006} C_VEL
LIN {X 0,Y 300.162,Z 232.541,A -85,B 0,C 180,E1 -16549.536,E2 -16549.536} C_VEL
LIN {X 0,Y 297.481,Z 230.011,A -85,B 0,C 180,E1 -16550.59,E2 -16550.59} C_VEL
LIN {X 0,Y 295.966,Z 227.142,A -85,B 0,C 180,E1 -16551.306,E2 -16551.306} C_VEL
LIN {X 0,Y 293.388,Z 225.277,A -85,B 0,C 180,E1 -16552.429,E2 -16552.429} C_VEL
LIN {X 0,Y 292.039,Z 222.873,A -85,B 0,C 180,E1 -16553.132,E2 -16553.132} C_VEL
LIN {X 0,Y 291.717,Z 221.456,A -85,B 0,C 180,E1 -16553.385,E2 -16553.385} C_VEL
LIN {X 0,Y 291.884,Z 221.436,A -85,B 0,C 180,E1 -16558.62,E2 -16558.62} C_VEL
LIN {X 0,Y 291.884,Z 221.438,A -85,B 0,C 180,E1 -16561.38,E2 -16561.38} C_VEL
LIN {X 0,Y 291.73,Z 221.46,A -85,B 0,C 180,E1 -16566.918,E2 -16566.918} C_VEL
LIN {X 0,Y 291.57,Z 221.48,A -85,B 0,C 180,E1 -16569.714,E2 -16569.714} C_VEL
LIN {X 0,Y 291.517,Z 221.479,A -85,B 0,C 180,E1 -16573.95,E2 -16573.95} C_VEL
LIN {X 0,Y 291.482,Z 221.484,A -85,B 0,C 180,E1 -16576.818,E2 -16576.818} C_VEL
LIN {X 0,Y 291.446,Z 221.491,A -85,B 0,C 180,E1 -16579.875,E2 -16579.875} C_VEL
LIN {X 0,Y 291.395,Z 221.495,A -85,B 0,C 180,E1 -16584.206,E2 -16584.206} C_VEL
LIN {X 0,Y 291.415,Z 221.494,A -85,B 0,C 180,E1 -16587.272,E2 -16587.272} C_VEL
LIN {X 0,Y 291.339,Z 221.518,A -85,B 0,C 180,E1 -16591.444,E2 -16591.444} C_VEL
LIN {X 0,Y 292.243,Z 224.168,A -85,B 0,C 180,E1 -16592.666,E2 -16592.666} C_VEL
LIN {X 0,Y 294.096,Z 226.245,A -85,B 0,C 180,E1 -16593.547,E2 -16593.547} C_VEL
LIN {X 0,Y 297.37,Z 230.306,A -85,B 0,C 180,E1 -16595.019,E2 -16595.019} C_VEL
LIN {X 0,Y 298.39,Z 231.695,A -85,B 0,C 180,E1 -16595.45,E2 -16595.45} C_VEL
LIN {X 0,Y 301.177,Z 235.366,A -85,B 0,C 180,E1 -16596.577,E2 -16596.577} C_VEL
LIN {X 0,Y 307.815,Z 244.644,A -85,B 0,C 180,E1 -16599.052,E2 -16599.052} C_VEL
LIN {X 0,Y 314.009,Z 253.902,A -85,B 0,C 180,E1 -16601.106,E2 -16601.106} C_VEL
LIN {X 0,Y 321.992,Z 267.036,A -85,B 0,C 180,E1 -16603.503,E2 -16603.503} C_VEL
LIN {X 0,Y 328.273,Z 278.494,A -85,B 0,C 180,E1 -16605.234,E2 -16605.234} C_VEL
LIN {X 0,Y 335.322,Z 293.149,A -85,B 0,C 180,E1 -16607.072,E2 -16607.072} C_VEL
LIN {X 0,Y 336.211,Z 295.103,A -85,B 0,C 180,E1 -16607.295,E2 -16607.295} C_VEL
LIN {X 0,Y 328.82,Z 434.134,A -85,B 0,C 180,E1 -16610.467,E2 -16610.467} C_VEL
LIN {X 0,Y 326.977,Z 451.439,A -85,B 0,C 180,E1 -16611.063,E2 -16611.063} C_VEL
LIN {X 0,Y 324.709,Z 466.975,A -85,B 0,C 180,E1 -16611.816,E2 -16611.816} C_VEL
LIN {X 0,Y 322.171,Z 481.647,A -85,B 0,C 180,E1 -16612.747,E2 -16612.747} C_VEL
LIN {X 0,Y 319.093,Z 496.345,A -85,B 0,C 180,E1 -16613.903,E2 -16613.903} C_VEL
LIN {X 0,Y 315.741,Z 510.393,A -85,B 0,C 180,E1 -16615.282,E2 -16615.282} C_VEL
LIN {X 0,Y 312.15,Z 524.072,A -85,B 0,C 180,E1 -16616.909,E2 -16616.909} C_VEL
LIN {X 0,Y 308.39,Z 537.133,A -85,B 0,C 180,E1 -16618.772,E2 -16618.772} C_VEL
LIN {X 0,Y 305.072,Z 548.339,A -85,B 0,C 180,E1 -16620.69,E2 -16620.69} C_VEL
LIN {X 0,Y 301.665,Z 559.555,A -85,B 0,C 180,E1 -16622.981,E2 -16622.981} C_VEL
LIN {X 0,Y 298.268,Z 570.454,A -85,B 0,C 180,E1 -16625.648,E2 -16625.648} C_VEL
LIN {X 0,Y 295.374,Z 579.867,A -85,B 0,C 180,E1 -16628.438,E2 -16628.438} C_VEL
LIN {X 0,Y 293.305,Z 587.363,A -85,B 0,C 180,E1 -16631.127,E2 -16631.127} C_VEL
LIN {X 0,Y 291.635,Z 593.716,A -85,B 0,C 180,E1 -16633.911,E2 -16633.911} C_VEL
LIN {X 0,Y 290.517,Z 598.953,A -85,B 0,C 180,E1 -16636.714,E2 -16636.714} C_VEL
LIN {X 0,Y 289.668,Z 603.922,A -85,B 0,C 180,E1 -16640.222,E2 -16640.222} C_VEL
LIN {X 0,Y 289.444,Z 606.676,A -85,B 0,C 180,E1 -16643.027,E2 -16643.027} C_VEL
LIN {X 0,Y 289.373,Z 608.508,A -85,B 0,C 180,E1 -16645.822,E2 -16645.822} C_VEL
LIN {X 0,Y 289.414,Z 609.283,A -85,B 0,C 180,E1 -16648.609,E2 -16648.609} C_VEL
LIN {X 0,Y 289.415,Z 609.146,A -85,B 0,C 180,E1 -16651.392,E2 -16651.392} C_VEL
LIN {X 0,Y 289.399,Z 607.944,A -85,B 0,C 180,E1 -16654.178,E2 -16654.178} C_VEL
LIN {X 0,Y 289.444,Z 605.801,A -85,B 0,C 180,E1 -16656.974,E2 -16656.974} C_VEL
LIN {X 0,Y 289.66,Z 602.558,A -85,B 0,C 180,E1 -16659.779,E2 -16659.779} C_VEL
LIN {X 0,Y 290.29,Z 598.264,A -85,B 0,C 180,E1 -16662.586,E2 -16662.586} C_VEL
LIN {X 0,Y 291.27,Z 592.811,A -85,B 0,C 180,E1 -16665.392,E2 -16665.392} C_VEL
LIN {X 0,Y 292.659,Z 586.05,A -85,B 0,C 180,E1 -16668.191,E2 -16668.191} C_VEL
LIN {X 0,Y 294.613,Z 577.928,A -85,B 0,C 180,E1 -16670.967,E2 -16670.967} C_VEL
LIN {X 0,Y 297.091,Z 568.215,A -85,B 0,C 180,E1 -16673.713,E2 -16673.713} C_VEL
LIN {X 0,Y 299.86,Z 558.138,A -85,B 0,C 180,E1 -16676.069,E2 -16676.069} C_VEL
LIN {X 0,Y 302.87,Z 546.297,A -85,B 0,C 180,E1 -16678.404,E2 -16678.404} C_VEL
LIN {X 0,Y 306.221,Z 533.361,A -85,B 0,C 180,E1 -16680.516,E2 -16680.516} C_VEL
LIN {X 0,Y 309.411,Z 520.534,A -85,B 0,C 180,E1 -16682.261,E2 -16682.261} C_VEL
LIN {X 0,Y 312.609,Z 506.165,A -85,B 0,C 180,E1 -16683.887,E2 -16683.887} C_VEL
LIN {X 0,Y 315.536,Z 491.84,A -85,B 0,C 180,E1 -16685.192,E2 -16685.192} C_VEL
LIN {X 0,Y 318.084,Z 476.642,A -85,B 0,C 180,E1 -16686.329,E2 -16686.329} C_VEL
LIN {X 0,Y 320.432,Z 459.943,A -85,B 0,C 180,E1 -16687.293,E2 -16687.293} C_VEL
LIN {X 0,Y 322.311,Z 443.791,A -85,B 0,C 180,E1 -16687.965,E2 -16687.965} C_VEL
LIN {X 0,Y 323.594,Z 427.164,A -85,B 0,C 180,E1 -16688.431,E2 -16688.431} C_VEL
LIN {X 0,Y 329.574,Z 292.998,A -85,B 0,C 180,E1 -16691.442,E2 -16691.442} C_VEL
LIN {X 0,Y 329.207,Z 291.402,A -85,B 0,C 180,E1 -16691.539,E2 -16691.539} C_VEL
LIN {X 0,Y 322.175,Z 276.766,A -85,B 0,C 180,E1 -16692.974,E2 -16692.974} C_VEL
LIN {X 0,Y 314.691,Z 262.288,A -85,B 0,C 180,E1 -16694.564,E2 -16694.564} C_VEL
LIN {X 0,Y 305.683,Z 246.564,A -85,B 0,C 180,E1 -16696.564,E2 -16696.564} C_VEL
LIN {X 0,Y 296.745,Z 232.039,A -85,B 0,C 180,E1 -16698.687,E2 -16698.687} C_VEL
LIN {X 0,Y 293.267,Z 226.58,A -85,B 0,C 180,E1 -16699.569,E2 -16699.569} C_VEL
LIN {X 0,Y 291.35,Z 221.508,A -85,B 0,C 180,E1 -16701.158,E2 -16701.158} C_VEL
LIN {X 0,Y 291.353,Z 221.491,A -85,B 0,C 180,E1 -16704.625,E2 -16704.625} C_VEL
LIN {X 0,Y 291.368,Z 221.481,A -85,B 0,C 180,E1 -16707.95,E2 -16707.95} C_VEL
LIN {X 0,Y 291.373,Z 221.505,A -85,B 0,C 180,E1 -16711.157,E2 -16711.157} C_VEL
LIN {X 0,Y 291.41,Z 221.47,A -85,B 0,C 180,E1 -16714.271,E2 -16714.271} C_VEL
LIN {X 0,Y 291.379,Z 221.504,A -85,B 0,C 180,E1 -16717.299,E2 -16717.299} C_VEL
LIN {X 0,Y 291.457,Z 221.458,A -85,B 0,C 180,E1 -16720.27,E2 -16720.27} C_VEL
LIN {X 0,Y 291.496,Z 221.488,A -85,B 0,C 180,E1 -16724.665,E2 -16724.665} C_VEL
LIN {X 0,Y 291.527,Z 221.442,A -85,B 0,C 180,E1 -16728.88,E2 -16728.88} C_VEL
LIN {X 0,Y 291.666,Z 221.463,A -85,B 0,C 180,E1 -16731.687,E2 -16731.687} C_VEL
LIN {X 0,Y 291.62,Z 221.455,A -85,B 0,C 180,E1 -16734.468,E2 -16734.468} C_VEL
LIN {X 0,Y 291.886,Z 221.401,A -85,B 0,C 180,E1 -16738.62,E2 -16738.62} C_VEL
LIN {X 0,Y 291.888,Z 221.438,A -85,B 0,C 180,E1 -16741.38,E2 -16741.38} C_VEL
LIN {X 0,Y 291.734,Z 221.447,A -85,B 0,C 180,E1 -16746.918,E2 -16746.918} C_VEL
LIN {X 0,Y 291.574,Z 221.47,A -85,B 0,C 180,E1 -16749.714,E2 -16749.714} C_VEL
LIN {X 0,Y 291.52,Z 221.474,A -85,B 0,C 180,E1 -16753.95,E2 -16753.95} C_VEL
LIN {X 0,Y 291.486,Z 221.48,A -85,B 0,C 180,E1 -16756.818,E2 -16756.818} C_VEL
LIN {X 0,Y 291.45,Z 221.471,A -85,B 0,C 180,E1 -16759.875,E2 -16759.875} C_VEL
LIN {X 0,Y 291.399,Z 221.483,A -85,B 0,C 180,E1 -16764.205,E2 -16764.205} C_VEL
LIN {X 0,Y 291.427,Z 221.487,A -85,B 0,C 180,E1 -16767.271,E2 -16767.271} C_VEL
LIN {X 0,Y 291.338,Z 221.498,A -85,B 0,C 180,E1 -16770.437,E2 -16770.437} C_VEL
LIN {X 0,Y 291.344,Z 221.496,A -85,B 0,C 180,E1 -16773.698,E2 -16773.698} C_VEL
LIN {X 0,Y 291.371,Z 221.486,A -85,B 0,C 180,E1 -16777.253,E2 -16777.253} C_VEL
LIN {X 0,Y 291.331,Z 221.507,A -85,B 0,C 180,E1 -16780.643,E2 -16780.643} C_VEL
LIN {X 0,Y 291.289,Z 221.497,A -85,B 0,C 180,E1 -16784.402,E2 -16784.402} C_VEL
LIN {X 0,Y 291.325,Z 221.494,A -85,B 0,C 180,E1 -16788.404,E2 -16788.404} C_VEL
LIN {X 0,Y 291.352,Z 221.505,A -85,B 0,C 180,E1 -16791.158,E2 -16791.158} C_VEL
LIN {X 0,Y 291.36,Z 221.489,A -85,B 0,C 180,E1 -16794.626,E2 -16794.626} C_VEL
LIN {X 0,Y 291.371,Z 221.491,A -85,B 0,C 180,E1 -16797.951,E2 -16797.951} C_VEL
LIN {X 0,Y 291.382,Z 221.502,A -85,B 0,C 180,E1 -16801.158,E2 -16801.158} C_VEL
LIN {X 0,Y 291.415,Z 221.498,A -85,B 0,C 180,E1 -16804.272,E2 -16804.272} C_VEL
LIN {X 0,Y 291.431,Z 221.541,A -85,B 0,C 180,E1 -16806.403,E2 -16806.403} C_VEL
LIN {X 0,Y 292.259,Z 224.067,A -85,B 0,C 180,E1 -16806.661,E2 -16806.661} C_VEL
LIN {X 0,Y 294.126,Z 226.252,A -85,B 0,C 180,E1 -16807.109,E2 -16807.109} C_VEL
LIN {X 0,Y 294.981,Z 227.595,A -85,B 0,C 180,E1 -16807.324,E2 -16807.324} C_VEL
LIN {X 0,Y 297.269,Z 230.72,A -85,B 0,C 180,E1 -16807.877,E2 -16807.877} C_VEL
LIN {X 0,Y 306.221,Z 243.825,A -85,B 0,C 180,E1 -16809.943,E2 -16809.943} C_VEL
LIN {X 0,Y 317.528,Z 261.707,A -85,B 0,C 180,E1 -16812.367,E2 -16812.367} C_VEL
LIN {X 0,Y 325.577,Z 275.989,A -85,B 0,C 180,E1 -16814,E2 -16814} C_VEL
LIN {X 0,Y 329.7,Z 284.378,A -85,B 0,C 180,E1 -16814.826,E2 -16814.826} C_VEL
LIN {X 0,Y 323.484,Z 419.403,A -85,B 0,C 180,E1 -16817.868,E2 -16817.868} C_VEL
LIN {X 0,Y 322.055,Z 435.827,A -85,B 0,C 180,E1 -16818.454,E2 -16818.454} C_VEL
LIN {X 0,Y 320.178,Z 451.684,A -85,B 0,C 180,E1 -16819.247,E2 -16819.247} C_VEL
LIN {X 0,Y 317.822,Z 467.608,A -85,B 0,C 180,E1 -16820.293,E2 -16820.293} C_VEL
LIN {X 0,Y 315.351,Z 482.228,A -85,B 0,C 180,E1 -16821.509,E2 -16821.509} C_VEL
LIN {X 0,Y 312.612,Z 495.523,A -85,B 0,C 180,E1 -16822.854,E2 -16822.854} C_VEL
LIN {X 0,Y 309.387,Z 509.848,A -85,B 0,C 180,E1 -16824.607,E2 -16824.607} C_VEL
LIN {X 0,Y 306.411,Z 521.988,A -85,B 0,C 180,E1 -16826.383,E2 -16826.383} C_VEL
LIN {X 0,Y 303.518,Z 533.255,A -85,B 0,C 180,E1 -16828.341,E2 -16828.341} C_VEL
LIN {X 0,Y 300.469,Z 544.515,A -85,B 0,C 180,E1 -16830.67,E2 -16830.67} C_VEL
LIN {X 0,Y 297.778,Z 554.183,A -85,B 0,C 180,E1 -16833.044,E2 -16833.044} C_VEL
LIN {X 0,Y 295.31,Z 563.543,A -85,B 0,C 180,E1 -16835.805,E2 -16835.805} C_VEL
LIN {X 0,Y 293.069,Z 572.245,A -85,B 0,C 180,E1 -16838.967,E2 -16838.967} C_VEL
LIN {X 0,Y 291.604,Z 578.531,A -85,B 0,C 180,E1 -16841.821,E2 -16841.821} C_VEL
LIN {X 0,Y 290.538,Z 583.464,A -85,B 0,C 180,E1 -16844.629,E2 -16844.629} C_VEL
LIN {X 0,Y 289.904,Z 586.665,A -85,B 0,C 180,E1 -16846.912,E2 -16846.912} C_VEL
LIN {X 0,Y 289.398,Z 589.761,A -85,B 0,C 180,E1 -16849.875,E2 -16849.875} C_VEL
LIN {X 0,Y 289.12,Z 591.799,A -85,B 0,C 180,E1 -16852.887,E2 -16852.887} C_VEL
LIN {X 0,Y 289.025,Z 592.637,A -85,B 0,C 180,E1 -16855.956,E2 -16855.956} C_VEL
LIN {X 0,Y 289.173,Z 592.35,A -85,B 0,C 180,E1 -16859.082,E2 -16859.082} C_VEL
LIN {X 0,Y 289.465,Z 590.855,A -85,B 0,C 180,E1 -16862.285,E2 -16862.285} C_VEL
LIN {X 0,Y 290.164,Z 587.962,A -85,B 0,C 180,E1 -16865.541,E2 -16865.541} C_VEL
LIN {X 0,Y 291.222,Z 583.6,A -85,B 0,C 180,E1 -16868.861,E2 -16868.861} C_VEL
LIN {X 0,Y 292.657,Z 578.294,A -85,B 0,C 180,E1 -16871.888,E2 -16871.888} C_VEL
LIN {X 0,Y 294.55,Z 571.787,A -85,B 0,C 180,E1 -16874.838,E2 -16874.838} C_VEL
LIN {X 0,Y 297.29,Z 563.121,A -85,B 0,C 180,E1 -16877.971,E2 -16877.971} C_VEL
LIN {X 0,Y 300.54,Z 553.23,A -85,B 0,C 180,E1 -16880.848,E2 -16880.848} C_VEL
LIN {X 0,Y 303.81,Z 543.029,A -85,B 0,C 180,E1 -16883.284,E2 -16883.284} C_VEL
LIN {X 0,Y 307.208,Z 532.242,A -85,B 0,C 180,E1 -16885.442,E2 -16885.442} C_VEL
LIN {X 0,Y 310.631,Z 520.862,A -85,B 0,C 180,E1 -16887.372,E2 -16887.372} C_VEL
LIN {X 0,Y 312.227,Z 515.316,A -85,B 0,C 180,E1 -16888.195,E2 -16888.195} C_VEL
LIN {X 0,Y 312.986,Z 510.854,A -85,B 0,C 180,E1 -16888.89,E2 -16888.89} C_VEL
LIN {X 0,Y 312.175,Z 497.771,A -85,B 0,C 180,E1 -16891.111,E2 -16891.111} C_VEL
LIN {X 0,Y 312.497,Z 493.035,A -85,B 0,C 180,E1 -16891.756,E2 -16891.756} C_VEL
LIN {X 0,Y 312.823,Z 491.381,A -85,B 0,C 180,E1 -16891.943,E2 -16891.943} C_VEL
LIN {X 0,Y 316.052,Z 477.212,A -85,B 0,C 180,E1 -16893.256,E2 -16893.256} C_VEL
LIN {X 0,Y 318.883,Z 462.307,A -85,B 0,C 180,E1 -16894.389,E2 -16894.389} C_VEL
LIN {X 0,Y 321.451,Z 445.738,A -85,B 0,C 180,E1 -16895.37,E2 -16895.37} C_VEL
LIN {X 0,Y 323.408,Z 429.796,A -85,B 0,C 180,E1 -16896.06,E2 -16896.06} C_VEL
LIN {X 0,Y 324.774,Z 412.803,A -85,B 0,C 180,E1 -16896.56,E2 -16896.56} C_VEL
LIN {X 0,Y 331.431,Z 290.944,A -85,B 0,C 180,E1 -16899.355,E2 -16899.355} C_VEL
LIN {X 0,Y 324.814,Z 277.985,A -85,B 0,C 180,E1 -16901.127,E2 -16901.127} C_VEL
LIN {X 0,Y 317.92,Z 266.879,A -85,B 0,C 180,E1 -16903.064,E2 -16903.064} C_VEL
LIN {X 0,Y 311.268,Z 256.933,A -85,B 0,C 180,E1 -16905.108,E2 -16905.108} C_VEL
LIN {X 0,Y 304.598,Z 247.809,A -85,B 0,C 180,E1 -16907.375,E2 -16907.375} C_VEL
LIN {X 0,Y 301.435,Z 243.629,A -85,B 0,C 180,E1 -16908.559,E2 -16908.559} C_VEL
LIN {X 0,Y 298.486,Z 239.944,A -85,B 0,C 180,E1 -16909.718,E2 -16909.718} C_VEL
LIN {X 0,Y 297.53,Z 238.693,A -85,B 0,C 180,E1 -16910.111,E2 -16910.111} C_VEL
LIN {X 0,Y 294.932,Z 235.844,A -85,B 0,C 180,E1 -16911.202,E2 -16911.202} C_VEL
LIN {X 0,Y 293.647,Z 233.607,A -85,B 0,C 180,E1 -16911.83,E2 -16911.83} C_VEL
LIN {X 0,Y 291.059,Z 231.291,A -85,B 0,C 180,E1 -16913.022,E2 -16913.022} C_VEL
LIN {X 0,Y 289.515,Z 228.353,A -85,B 0,C 180,E1 -16913.869,E2 -16913.869} C_VEL
LIN {X 0,Y 286.294,Z 226.247,A -85,B 0,C 180,E1 -16915.512,E2 -16915.512} C_VEL
LIN {X 0,Y 285.02,Z 224.112,A -85,B 0,C 180,E1 -16916.333,E2 -16916.333} C_VEL
LIN {X 0,Y 284.635,Z 222.343,A -85,B 0,C 180,E1 -16916.727,E2 -16916.727} C_VEL
LIN {X 0,Y 284.918,Z 222.304,A -85,B 0,C 180,E1 -16920,E2 -16920} C_VEL
LIN {X 0,Y 284.737,Z 222.324,A -85,B 0,C 180,E1 -16922.83,E2 -16922.83} C_VEL
LIN {X 0,Y 284.681,Z 222.338,A -85,B 0,C 180,E1 -16927.09,E2 -16927.09} C_VEL
LIN {X 0,Y 284.514,Z 222.358,A -85,B 0,C 180,E1 -16929.957,E2 -16929.957} C_VEL
LIN {X 0,Y 284.476,Z 222.357,A -85,B 0,C 180,E1 -16934.303,E2 -16934.303} C_VEL
LIN {X 0,Y 284.42,Z 222.366,A -85,B 0,C 180,E1 -16937.249,E2 -16937.249} C_VEL
LIN {X 0,Y 284.374,Z 222.376,A -85,B 0,C 180,E1 -16940.242,E2 -16940.242} C_VEL
LIN {X 0,Y 284.364,Z 222.371,A -85,B 0,C 180,E1 -16943.875,E2 -16943.875} C_VEL
LIN {X 0,Y 284.39,Z 222.369,A -85,B 0,C 180,E1 -16947.173,E2 -16947.173} C_VEL
LIN {X 0,Y 284.356,Z 222.53,A -85,B 0,C 180,E1 -16948.611,E2 -16948.611} C_VEL
LIN {X 0,Y 284.607,Z 223.577,A -85,B 0,C 180,E1 -16949.038,E2 -16949.038} C_VEL
LIN {X 0,Y 285.735,Z 225.81,A -85,B 0,C 180,E1 -16949.803,E2 -16949.803} C_VEL
LIN {X 0,Y 287.974,Z 227.753,A -85,B 0,C 180,E1 -16951.035,E2 -16951.035} C_VEL
LIN {X 0,Y 290.008,Z 230.266,A -85,B 0,C 180,E1 -16952.1,E2 -16952.1} C_VEL
LIN {X 0,Y 292.92,Z 233.957,A -85,B 0,C 180,E1 -16953.536,E2 -16953.536} C_VEL
LIN {X 0,Y 295.965,Z 237.782,A -85,B 0,C 180,E1 -16954.921,E2 -16954.921} C_VEL
LIN {X 0,Y 298.773,Z 241.552,A -85,B 0,C 180,E1 -16956.095,E2 -16956.095} C_VEL
LIN {X 0,Y 305.151,Z 250.704,A -85,B 0,C 180,E1 -16958.56,E2 -16958.56} C_VEL
LIN {X 0,Y 311.199,Z 259.975,A -85,B 0,C 180,E1 -16960.638,E2 -16960.638} C_VEL
LIN {X 0,Y 318.896,Z 272.91,A -85,B 0,C 180,E1 -16963.028,E2 -16963.028} C_VEL
LIN {X 0,Y 325.668,Z 285.842,A -85,B 0,C 180,E1 -16964.964,E2 -16964.964} C_VEL
LIN {X 0,Y 331.197,Z 297.71,A -85,B 0,C 180,E1 -16966.463,E2 -16966.463} C_VEL
LIN {X 0,Y 325.009,Z 410.065,A -85,B 0,C 180,E1 -16969.023,E2 -16969.023} C_VEL
LIN {X 0,Y 323.477,Z 436.194,A -85,B 0,C 180,E1 -16969.681,E2 -16969.681} C_VEL
LIN {X 0,Y 321.504,Z 453.181,A -85,B 0,C 180,E1 -16970.29,E2 -16970.29} C_VEL
LIN {X 0,Y 318.984,Z 469.222,A -85,B 0,C 180,E1 -16971.104,E2 -16971.104} C_VEL
LIN {X 0,Y 316.148,Z 484.263,A -85,B 0,C 180,E1 -16972.114,E2 -16972.114} C_VEL
LIN {X 0,Y 312.625,Z 500.004,A -85,B 0,C 180,E1 -16973.436,E2 -16973.436} C_VEL
LIN {X 0,Y 308.907,Z 514.786,A -85,B 0,C 180,E1 -16974.989,E2 -16974.989} C_VEL
LIN {X 0,Y 305.202,Z 527.883,A -85,B 0,C 180,E1 -16976.649,E2 -16976.649} C_VEL
LIN {X 0,Y 301.73,Z 539.295,A -85,B 0,C 180,E1 -16978.395,E2 -16978.395} C_VEL
LIN {X 0,Y 297.752,Z 551.875,A -85,B 0,C 180,E1 -16980.686,E2 -16980.686} C_VEL
LIN {X 0,Y 294.3,Z 562.56,A -85,B 0,C 180,E1 -16983.018,E2 -16983.018} C_VEL
LIN {X 0,Y 290.922,Z 572.962,A -85,B 0,C 180,E1 -16985.753,E2 -16985.753} C_VEL
LIN {X 0,Y 288.162,Z 581.669,A -85,B 0,C 180,E1 -16988.542,E2 -16988.542} C_VEL
LIN {X 0,Y 286.006,Z 588.985,A -85,B 0,C 180,E1 -16991.371,E2 -16991.371} C_VEL
LIN {X 0,Y 284.191,Z 595.89,A -85,B 0,C 180,E1 -16994.679,E2 -16994.679} C_VEL
LIN {X 0,Y 283.11,Z 601.018,A -85,B 0,C 180,E1 -16997.819,E2 -16997.819} C_VEL
LIN {X 0,Y 282.431,Z 605.277,A -85,B 0,C 180,E1 -17001.414,E2 -17001.414} C_VEL
LIN {X 0,Y 282.326,Z 607.772,A -85,B 0,C 180,E1 -17004.7,E2 -17004.7} C_VEL
LIN {X 0,Y 282.327,Z 608.835,A -85,B 0,C 180,E1 -17007.147,E2 -17007.147} C_VEL
LIN {X 0,Y 282.355,Z 609.113,A -85,B 0,C 180,E1 -17010,E2 -17010} C_VEL
LIN {X 0,Y 282.335,Z 608.449,A -85,B 0,C 180,E1 -17012.854,E2 -17012.854} C_VEL
LIN {X 0,Y 282.334,Z 606.735,A -85,B 0,C 180,E1 -17015.715,E2 -17015.715} C_VEL
LIN {X 0,Y 282.427,Z 604.056,A -85,B 0,C 180,E1 -17018.587,E2 -17018.587} C_VEL
LIN {X 0,Y 282.849,Z 600.237,A -85,B 0,C 180,E1 -17021.466,E2 -17021.466} C_VEL
LIN {X 0,Y 283.765,Z 595.375,A -85,B 0,C 180,E1 -17024.34,E2 -17024.34} C_VEL
LIN {X 0,Y 284.951,Z 589.224,A -85,B 0,C 180,E1 -17027.216,E2 -17027.216} C_VEL
LIN {X 0,Y 286.812,Z 581.77,A -85,B 0,C 180,E1 -17030.063,E2 -17030.063} C_VEL
LIN {X 0,Y 289.061,Z 572.834,A -85,B 0,C 180,E1 -17032.893,E2 -17032.893} C_VEL
LIN {X 0,Y 292.031,Z 562.166,A -85,B 0,C 180,E1 -17035.67,E2 -17035.67} C_VEL
LIN {X 0,Y 294.934,Z 551.905,A -85,B 0,C 180,E1 -17037.886,E2 -17037.886} C_VEL
LIN {X 0,Y 298.125,Z 539.992,A -85,B 0,C 180,E1 -17040.063,E2 -17040.063} C_VEL
LIN {X 0,Y 301.466,Z 527.11,A -85,B 0,C 180,E1 -17042.03,E2 -17042.03} C_VEL
LIN {X 0,Y 304.584,Z 514.57,A -85,B 0,C 180,E1 -17043.627,E2 -17043.627} C_VEL
LIN {X 0,Y 307.887,Z 499.594,A -85,B 0,C 180,E1 -17045.196,E2 -17045.196} C_VEL
LIN {X 0,Y 310.689,Z 485.12,A -85,B 0,C 180,E1 -17046.427,E2 -17046.427} C_VEL
LIN {X 0,Y 313.253,Z 469.55,A -85,B 0,C 180,E1 -17047.486,E2 -17047.486} C_VEL
LIN {X 0,Y 315.355,Z 453.906,A -85,B 0,C 180,E1 -17048.304,E2 -17048.304} C_VEL
LIN {X 0,Y 317.154,Z 437.147,A -85,B 0,C 180,E1 -17048.904,E2 -17048.904} C_VEL
LIN {X 0,Y 318.474,Z 411.231,A -85,B 0,C 180,E1 -17049.546,E2 -17049.546} C_VEL
LIN {X 0,Y 323.97,Z 294.602,A -85,B 0,C 180,E1 -17052.183,E2 -17052.183} C_VEL
LIN {X 0,Y 315.775,Z 277.526,A -85,B 0,C 180,E1 -17053.918,E2 -17053.918} C_VEL
LIN {X 0,Y 308.06,Z 262.921,A -85,B 0,C 180,E1 -17055.623,E2 -17055.623} C_VEL
LIN {X 0,Y 300.555,Z 249.896,A -85,B 0,C 180,E1 -17057.36,E2 -17057.36} C_VEL
LIN {X 0,Y 292.373,Z 236.555,A -85,B 0,C 180,E1 -17059.371,E2 -17059.371} C_VEL
LIN {X 0,Y 285.719,Z 226.168,A -85,B 0,C 180,E1 -17061.153,E2 -17061.153} C_VEL
LIN {X 0,Y 284.301,Z 222.462,A -85,B 0,C 180,E1 -17062.333,E2 -17062.333} C_VEL
LIN {X 0,Y 284.306,Z 222.379,A -85,B 0,C 180,E1 -17065.351,E2 -17065.351} C_VEL
LIN {X 0,Y 284.292,Z 222.361,A -85,B 0,C 180,E1 -17068.725,E2 -17068.725} C_VEL
LIN {X 0,Y 284.391,Z 222.352,A -85,B 0,C 180,E1 -17072.829,E2 -17072.829} C_VEL
LIN {X 0,Y 284.365,Z 222.375,A -85,B 0,C 180,E1 -17076.707,E2 -17076.707} C_VEL
LIN {X 0,Y 284.375,Z 222.342,A -85,B 0,C 180,E1 -17079.904,E2 -17079.904} C_VEL
LIN {X 0,Y 284.445,Z 222.368,A -85,B 0,C 180,E1 -17084.492,E2 -17084.492} C_VEL
LIN {X 0,Y 284.464,Z 222.32,A -85,B 0,C 180,E1 -17088.601,E2 -17088.601} C_VEL
LIN {X 0,Y 284.62,Z 222.34,A -85,B 0,C 180,E1 -17091.48,E2 -17091.48} C_VEL
LIN {X 0,Y 284.59,Z 222.332,A -85,B 0,C 180,E1 -17094.331,E2 -17094.331} C_VEL
LIN {X 0,Y 284.852,Z 222.275,A -85,B 0,C 180,E1 -17098.586,E2 -17098.586} C_VEL
LIN {X 0,Y 284.854,Z 222.314,A -85,B 0,C 180,E1 -17101.414,E2 -17101.414} C_VEL
LIN {X 0,Y 284.685,Z 222.327,A -85,B 0,C 180,E1 -17107.09,E2 -17107.09} C_VEL
LIN {X 0,Y 284.518,Z 222.346,A -85,B 0,C 180,E1 -17109.957,E2 -17109.957} C_VEL
LIN {X 0,Y 284.48,Z 222.355,A -85,B 0,C 180,E1 -17114.303,E2 -17114.303} C_VEL
LIN {X 0,Y 284.424,Z 222.351,A -85,B 0,C 180,E1 -17117.248,E2 -17117.248} C_VEL
LIN {X 0,Y 284.378,Z 222.356,A -85,B 0,C 180,E1 -17120.242,E2 -17120.242} C_VEL
LIN {X 0,Y 284.368,Z 222.362,A -85,B 0,C 180,E1 -17123.875,E2 -17123.875} C_VEL
LIN {X 0,Y 284.365,Z 222.373,A -85,B 0,C 180,E1 -17128.007,E2 -17128.007} C_VEL
LIN {X 0,Y 284.295,Z 222.364,A -85,B 0,C 180,E1 -17131.274,E2 -17131.274} C_VEL
LIN {X 0,Y 284.34,Z 222.38,A -85,B 0,C 180,E1 -17135.348,E2 -17135.348} C_VEL
LIN {X 0,Y 284.307,Z 222.361,A -85,B 0,C 180,E1 -17138.17,E2 -17138.17} C_VEL
LIN {X 0,Y 284.269,Z 222.383,A -85,B 0,C 180,E1 -17142.124,E2 -17142.124} C_VEL
LIN {X 0,Y 284.255,Z 222.39,A -85,B 0,C 180,E1 -17146.189,E2 -17146.189} C_VEL
LIN {X 0,Y 284.306,Z 222.371,A -85,B 0,C 180,E1 -17150.024,E2 -17150.024} C_VEL
LIN {X 0,Y 284.332,Z 222.362,A -85,B 0,C 180,E1 -17153.614,E2 -17153.614} C_VEL
LIN {X 0,Y 284.307,Z 222.378,A -85,B 0,C 180,E1 -17157.19,E2 -17157.19} C_VEL
LIN {X 0,Y 284.358,Z 222.378,A -85,B 0,C 180,E1 -17160.376,E2 -17160.376} C_VEL
LIN {X 0,Y 284.378,Z 222.375,A -85,B 0,C 180,E1 -17164.374,E2 -17164.374} C_VEL
LIN {X 0,Y 284.348,Z 222.376,A -85,B 0,C 180,E1 -17164.959,E2 -17164.959} C_VEL
LIN {X 0,Y 285.297,Z 225.107,A -85,B 0,C 180,E1 -17165.271,E2 -17165.271} C_VEL
LIN {X 0,Y 287.171,Z 227.175,A -85,B 0,C 180,E1 -17165.743,E2 -17165.743} C_VEL
LIN {X 0,Y 289.913,Z 231.292,A -85,B 0,C 180,E1 -17166.457,E2 -17166.457} C_VEL
LIN {X 0,Y 291.078,Z 232.783,A -85,B 0,C 180,E1 -17166.745,E2 -17166.745} C_VEL
LIN {X 0,Y 300.621,Z 246.586,A -85,B 0,C 180,E1 -17169.048,E2 -17169.048} C_VEL
LIN {X 0,Y 311.477,Z 263.62,A -85,B 0,C 180,E1 -17171.465,E2 -17171.465} C_VEL
LIN {X 0,Y 320.504,Z 279.481,A -85,B 0,C 180,E1 -17173.363,E2 -17173.363} C_VEL
LIN {X 0,Y 324.071,Z 286.655,A -85,B 0,C 180,E1 -17174.098,E2 -17174.098} C_VEL
LIN {X 0,Y 317.711,Z 419.705,A -85,B 0,C 180,E1 -17177.135,E2 -17177.135} C_VEL
LIN {X 0,Y 316.21,Z 436.468,A -85,B 0,C 180,E1 -17177.745,E2 -17177.745} C_VEL
LIN {X 0,Y 314.247,Z 452.296,A -85,B 0,C 180,E1 -17178.551,E2 -17178.551} C_VEL
LIN {X 0,Y 311.813,Z 468.143,A -85,B 0,C 180,E1 -17179.612,E2 -17179.612} C_VEL
LIN {X 0,Y 309.277,Z 482.701,A -85,B 0,C 180,E1 -17180.847,E2 -17180.847} C_VEL
LIN {X 0,Y 306.401,Z 496.187,A -85,B 0,C 180,E1 -17182.235,E2 -17182.235} C_VEL
LIN {X 0,Y 303.212,Z 509.907,A -85,B 0,C 180,E1 -17183.946,E2 -17183.946} C_VEL
LIN {X 0,Y 299.768,Z 523.358,A -85,B 0,C 180,E1 -17185.966,E2 -17185.966} C_VEL
LIN {X 0,Y 296.79,Z 534.52,A -85,B 0,C 180,E1 -17187.964,E2 -17187.964} C_VEL
LIN {X 0,Y 293.633,Z 545.627,A -85,B 0,C 180,E1 -17190.342,E2 -17190.342} C_VEL
LIN {X 0,Y 290.873,Z 555.141,A -85,B 0,C 180,E1 -17192.769,E2 -17192.769} C_VEL
LIN {X 0,Y 288.327,Z 564.37,A -85,B 0,C 180,E1 -17195.595,E2 -17195.595} C_VEL
LIN {X 0,Y 286.248,Z 572.121,A -85,B 0,C 180,E1 -17198.471,E2 -17198.471} C_VEL
LIN {X 0,Y 284.682,Z 578.445,A -85,B 0,C 180,E1 -17201.39,E2 -17201.39} C_VEL
LIN {X 0,Y 283.537,Z 583.577,A -85,B 0,C 180,E1 -17204.351,E2 -17204.351} C_VEL
LIN {X 0,Y 282.71,Z 587.619,A -85,B 0,C 180,E1 -17207.356,E2 -17207.356} C_VEL
LIN {X 0,Y 282.232,Z 590.455,A -85,B 0,C 180,E1 -17210.402,E2 -17210.402} C_VEL
LIN {X 0,Y 281.976,Z 592.235,A -85,B 0,C 180,E1 -17213.502,E2 -17213.502} C_VEL
LIN {X 0,Y 281.931,Z 592.924,A -85,B 0,C 180,E1 -17216.66,E2 -17216.66} C_VEL
LIN {X 0,Y 282.106,Z 592.35,A -85,B 0,C 180,E1 -17219.884,E2 -17219.884} C_VEL
LIN {X 0,Y 282.535,Z 590.551,A -85,B 0,C 180,E1 -17223.177,E2 -17223.177} C_VEL
LIN {X 0,Y 283.338,Z 587.408,A -85,B 0,C 180,E1 -17226.533,E2 -17226.533} C_VEL
LIN {X 0,Y 284.598,Z 582.77,A -85,B 0,C 180,E1 -17229.944,E2 -17229.944} C_VEL
LIN {X 0,Y 286.476,Z 576.464,A -85,B 0,C 180,E1 -17233.385,E2 -17233.385} C_VEL
LIN {X 0,Y 288.739,Z 569.394,A -85,B 0,C 180,E1 -17236.395,E2 -17236.395} C_VEL
LIN {X 0,Y 291.641,Z 560.654,A -85,B 0,C 180,E1 -17239.41,E2 -17239.41} C_VEL
LIN {X 0,Y 294.671,Z 551.849,A -85,B 0,C 180,E1 -17241.91,E2 -17241.91} C_VEL
LIN {X 0,Y 298.327,Z 541.279,A -85,B 0,C 180,E1 -17244.411,E2 -17244.411} C_VEL
LIN {X 0,Y 302.269,Z 528.969,A -85,B 0,C 180,E1 -17246.826,E2 -17246.826} C_VEL
LIN {X 0,Y 306.194,Z 516.242,A -85,B 0,C 180,E1 -17248.863,E2 -17248.863} C_VEL
LIN {X 0,Y 309.697,Z 503.639,A -85,B 0,C 180,E1 -17250.555,E2 -17250.555} C_VEL
LIN {X 0,Y 312.823,Z 491.381,A -85,B 0,C 180,E1 -17251.943,E2 -17251.943} C_VEL
LIN {X 0,Y 313.473,Z 486.444,A -85,B 0,C 180,E1 -17252.529,E2 -17252.529} C_VEL
LIN {X 0,Y 312.674,Z 472.001,A -85,B 0,C 180,E1 -17254.446,E2 -17254.446} C_VEL
LIN {X 0,Y 312.906,Z 466.81,A -85,B 0,C 180,E1 -17254.957,E2 -17254.957} C_VEL
LIN {X 0,Y 313.171,Z 465.007,A -85,B 0,C 180,E1 -17255.092,E2 -17255.092} C_VEL
LIN {X 0,Y 315.762,Z 449.563,A -85,B 0,C 180,E1 -17256.065,E2 -17256.065} C_VEL
LIN {X 0,Y 317.949,Z 433.216,A -85,B 0,C 180,E1 -17256.817,E2 -17256.817} C_VEL
LIN {X 0,Y 319.471,Z 416.692,A -85,B 0,C 180,E1 -17257.349,E2 -17257.349} C_VEL
LIN {X 0,Y 326.555,Z 293.786,A -85,B 0,C 180,E1 -17260.213,E2 -17260.213} C_VEL
LIN {X 0,Y 320.764,Z 282.452,A -85,B 0,C 180,E1 -17261.828,E2 -17261.828} C_VEL
LIN {X 0,Y 314.097,Z 271.491,A -85,B 0,C 180,E1 -17263.791,E2 -17263.791} C_VEL
LIN {X 0,Y 307.943,Z 262.279,A -85,B 0,C 180,E1 -17265.767,E2 -17265.767} C_VEL
LIN {X 0,Y 302.024,Z 253.891,A -85,B 0,C 180,E1 -17267.869,E2 -17267.869} C_VEL
LIN {X 0,Y 298.707,Z 249.525,A -85,B 0,C 180,E1 -17269.151,E2 -17269.151} C_VEL
LIN {X 0,Y 295.819,Z 245.689,A -85,B 0,C 180,E1 -17270.337,E2 -17270.337} C_VEL
LIN {X 0,Y 292.426,Z 241.629,A -85,B 0,C 180,E1 -17271.839,E2 -17271.839} C_VEL
LIN {X 0,Y 291.341,Z 239.945,A -85,B 0,C 180,E1 -17272.376,E2 -17272.376} C_VEL
LIN {X 0,Y 288.732,Z 237.296,A -85,B 0,C 180,E1 -17273.638,E2 -17273.638} C_VEL
LIN {X 0,Y 287.401,Z 234.861,A -85,B 0,C 180,E1 -17274.387,E2 -17274.387} C_VEL
LIN {X 0,Y 284.682,Z 232.967,A -85,B 0,C 180,E1 -17275.841,E2 -17275.841} C_VEL
LIN {X 0,Y 283.03,Z 230.3,A -85,B 0,C 180,E1 -17276.931,E2 -17276.931} C_VEL
LIN {X 0,Y 282.472,Z 229.034,A -85,B 0,C 180,E1 -17277.344,E2 -17277.344} C_VEL
LIN {X 0,Y 279.909,Z 227.405,A -85,B 0,C 180,E1 -17279.011,E2 -17279.011} C_VEL
LIN {X 0,Y 278.221,Z 224.777,A -85,B 0,C 180,E1 -17280.452,E2 -17280.452} C_VEL
LIN {X 0,Y 277.827,Z 223.186,A -85,B 0,C 180,E1 -17280.996,E2 -17280.996} C_VEL
LIN {X 0,Y 277.457,Z 223.238,A -85,B 0,C 180,E1 -17284.358,E2 -17284.358} C_VEL
LIN {X 0,Y 277.636,Z 223.215,A -85,B 0,C 180,E1 -17287.271,E2 -17287.271} C_VEL
LIN {X 0,Y 277.456,Z 223.234,A -85,B 0,C 180,E1 -17290.213,E2 -17290.213} C_VEL
LIN {X 0,Y 277.43,Z 223.237,A -85,B 0,C 180,E1 -17294.674,E2 -17294.674} C_VEL
LIN {X 0,Y 277.34,Z 223.245,A -85,B 0,C 180,E1 -17299.234,E2 -17299.234} C_VEL
LIN {X 0,Y 277.314,Z 223.249,A -85,B 0,C 180,E1 -17304.17,E2 -17304.17} C_VEL
LIN {X 0,Y 277.353,Z 223.559,A -85,B 0,C 180,E1 -17304.383,E2 -17304.383} C_VEL
LIN {X 0,Y 278.156,Z 225.881,A -85,B 0,C 180,E1 -17305.249,E2 -17305.249} C_VEL
LIN {X 0,Y 280.45,Z 228.277,A -85,B 0,C 180,E1 -17307.033,E2 -17307.033} C_VEL
LIN {X 0,Y 282.47,Z 229.354,A -85,B 0,C 180,E1 -17308.313,E2 -17308.313} C_VEL
LIN {X 0,Y 283.691,Z 231.949,A -85,B 0,C 180,E1 -17309.191,E2 -17309.191} C_VEL
LIN {X 0,Y 285.915,Z 234.231,A -85,B 0,C 180,E1 -17310.508,E2 -17310.508} C_VEL
LIN {X 0,Y 287.021,Z 235.336,A -85,B 0,C 180,E1 -17311.104,E2 -17311.104} C_VEL
LIN {X 0,Y 291.248,Z 240.915,A -85,B 0,C 180,E1 -17313.279,E2 -17313.279} C_VEL
LIN {X 0,Y 293.58,Z 243.876,A -85,B 0,C 180,E1 -17314.376,E2 -17314.376} C_VEL
LIN {X 0,Y 296.54,Z 247.915,A -85,B 0,C 180,E1 -17315.666,E2 -17315.666} C_VEL
LIN {X 0,Y 302.394,Z 256.574,A -85,B 0,C 180,E1 -17318.008,E2 -17318.008} C_VEL
LIN {X 0,Y 308.128,Z 265.616,A -85,B 0,C 180,E1 -17320.063,E2 -17320.063} C_VEL
LIN {X 0,Y 315.236,Z 277.825,A -85,B 0,C 180,E1 -17322.368,E2 -17322.368} C_VEL
LIN {X 0,Y 321.702,Z 290.356,A -85,B 0,C 180,E1 -17324.301,E2 -17324.301} C_VEL
LIN {X 0,Y 326.332,Z 300.37,A -85,B 0,C 180,E1 -17325.607,E2 -17325.607} C_VEL
LIN {X 0,Y 318.57,Z 434.09,A -85,B 0,C 180,E1 -17328.728,E2 -17328.728} C_VEL
LIN {X 0,Y 316.595,Z 451.265,A -85,B 0,C 180,E1 -17329.332,E2 -17329.332} C_VEL
LIN {X 0,Y 313.974,Z 467.784,A -85,B 0,C 180,E1 -17330.154,E2 -17330.154} C_VEL
LIN {X 0,Y 311.064,Z 483.099,A -85,B 0,C 180,E1 -17331.174,E2 -17331.174} C_VEL
LIN {X 0,Y 307.349,Z 498.993,A -85,B 0,C 180,E1 -17332.497,E2 -17332.497} C_VEL
LIN {X 0,Y 303.565,Z 513.563,A -85,B 0,C 180,E1 -17334.024,E2 -17334.024} C_VEL
LIN {X 0,Y 299.281,Z 528.172,A -85,B 0,C 180,E1 -17335.9,E2 -17335.9} C_VEL
LIN {X 0,Y 295.093,Z 541.464,A -85,B 0,C 180,E1 -17338.001,E2 -17338.001} C_VEL
LIN {X 0,Y 291.202,Z 553.023,A -85,B 0,C 180,E1 -17340.204,E2 -17340.204} C_VEL
LIN {X 0,Y 287.438,Z 564.001,A -85,B 0,C 180,E1 -17342.714,E2 -17342.714} C_VEL
LIN {X 0,Y 283.98,Z 574.127,A -85,B 0,C 180,E1 -17345.511,E2 -17345.511} C_VEL
LIN {X 0,Y 281.438,Z 581.654,A -85,B 0,C 180,E1 -17348.003,E2 -17348.003} C_VEL
LIN {X 0,Y 279.195,Z 588.931,A -85,B 0,C 180,E1 -17350.899,E2 -17350.899} C_VEL
LIN {X 0,Y 277.462,Z 594.998,A -85,B 0,C 180,E1 -17353.822,E2 -17353.822} C_VEL
LIN {X 0,Y 276.118,Z 600.904,A -85,B 0,C 180,E1 -17357.506,E2 -17357.506} C_VEL
LIN {X 0,Y 275.362,Z 605.131,A -85,B 0,C 180,E1 -17361.192,E2 -17361.192} C_VEL
LIN {X 0,Y 275.226,Z 607.732,A -85,B 0,C 180,E1 -17364.794,E2 -17364.794} C_VEL
LIN {X 0,Y 275.235,Z 608.65,A -85,B 0,C 180,E1 -17367.073,E2 -17367.073} C_VEL
LIN {X 0,Y 275.277,Z 608.9,A -85,B 0,C 180,E1 -17370,E2 -17370} C_VEL
LIN {X 0,Y 275.244,Z 608.222,A -85,B 0,C 180,E1 -17372.928,E2 -17372.928} C_VEL
LIN {X 0,Y 275.229,Z 606.477,A -85,B 0,C 180,E1 -17375.863,E2 -17375.863} C_VEL
LIN {X 0,Y 275.358,Z 603.782,A -85,B 0,C 180,E1 -17378.809,E2 -17378.809} C_VEL
LIN {X 0,Y 276.054,Z 598.845,A -85,B 0,C 180,E1 -17382.498,E2 -17382.498} C_VEL
LIN {X 0,Y 277.092,Z 593.546,A -85,B 0,C 180,E1 -17385.462,E2 -17385.462} C_VEL
LIN {X 0,Y 278.509,Z 587.13,A -85,B 0,C 180,E1 -17388.387,E2 -17388.387} C_VEL
LIN {X 0,Y 280.536,Z 579.305,A -85,B 0,C 180,E1 -17391.3,E2 -17391.3} C_VEL
LIN {X 0,Y 283.162,Z 569.875,A -85,B 0,C 180,E1 -17394.175,E2 -17394.175} C_VEL
LIN {X 0,Y 286.002,Z 560.153,A -85,B 0,C 180,E1 -17396.645,E2 -17396.645} C_VEL
LIN {X 0,Y 288.865,Z 549.974,A -85,B 0,C 180,E1 -17398.853,E2 -17398.853} C_VEL
LIN {X 0,Y 292.427,Z 537.382,A -85,B 0,C 180,E1 -17401.112,E2 -17401.112} C_VEL
LIN {X 0,Y 296.006,Z 524.006,A -85,B 0,C 180,E1 -17403.099,E2 -17403.099} C_VEL
LIN {X 0,Y 299.594,Z 509.457,A -85,B 0,C 180,E1 -17404.875,E2 -17404.875} C_VEL
LIN {X 0,Y 302.756,Z 495.233,A -85,B 0,C 180,E1 -17406.295,E2 -17406.295} C_VEL
LIN {X 0,Y 305.688,Z 479.93,A -85,B 0,C 180,E1 -17407.535,E2 -17407.535} C_VEL
LIN {X 0,Y 308.347,Z 462.916,A -85,B 0,C 180,E1 -17408.605,E2 -17408.605} C_VEL
LIN {X 0,Y 310.424,Z 446.608,A -85,B 0,C 180,E1 -17409.34,E2 -17409.34} C_VEL
LIN {X 0,Y 311.919,Z 430.143,A -85,B 0,C 180,E1 -17409.848,E2 -17409.848} C_VEL
LIN {X 0,Y 318.291,Z 296.795,A -85,B 0,C 180,E1 -17412.945,E2 -17412.945} C_VEL
LIN {X 0,Y 308.589,Z 276.734,A -85,B 0,C 180,E1 -17415.089,E2 -17415.089} C_VEL
LIN {X 0,Y 299.907,Z 260.697,A -85,B 0,C 180,E1 -17417.107,E2 -17417.107} C_VEL
LIN {X 0,Y 288.883,Z 242.261,A -85,B 0,C 180,E1 -17419.857,E2 -17419.857} C_VEL
LIN {X 0,Y 280.999,Z 230.338,A -85,B 0,C 180,E1 -17421.976,E2 -17421.976} C_VEL
LIN {X 0,Y 278.224,Z 225.965,A -85,B 0,C 180,E1 -17422.794,E2 -17422.794} C_VEL
LIN {X 0,Y 277.295,Z 223.236,A -85,B 0,C 180,E1 -17423.717,E2 -17423.717} C_VEL
LIN {X 0,Y 277.242,Z 223.24,A -85,B 0,C 180,E1 -17427.836,E2 -17427.836} C_VEL
LIN {X 0,Y 277.283,Z 223.26,A -85,B 0,C 180,E1 -17431.212,E2 -17431.212} C_VEL
LIN {X 0,Y 277.31,Z 223.225,A -85,B 0,C 180,E1 -17434.479,E2 -17434.479} C_VEL
LIN {X 0,Y 277.281,Z 223.26,A -85,B 0,C 180,E1 -17437.655,E2 -17437.655} C_VEL
LIN {X 0,Y 277.319,Z 223.217,A -85,B 0,C 180,E1 -17440.764,E2 -17440.764} C_VEL
LIN {X 0,Y 277.408,Z 223.238,A -85,B 0,C 180,E1 -17445.325,E2 -17445.325} C_VEL
LIN {X 0,Y 277.453,Z 223.202,A -85,B 0,C 180,E1 -17449.787,E2 -17449.787} C_VEL
LIN {X 0,Y 277.626,Z 223.215,A -85,B 0,C 180,E1 -17452.728,E2 -17452.728} C_VEL
LIN {X 0,Y 277.818,Z 223.15,A -85,B 0,C 180,E1 -17458.55,E2 -17458.55} C_VEL
LIN {X 0,Y 277.82,Z 223.191,A -85,B 0,C 180,E1 -17461.45,E2 -17461.45} C_VEL
LIN {X 0,Y 277.64,Z 223.208,A -85,B 0,C 180,E1 -17467.271,E2 -17467.271} C_VEL
LIN {X 0,Y 277.46,Z 223.222,A -85,B 0,C 180,E1 -17470.213,E2 -17470.213} C_VEL
LIN {X 0,Y 277.433,Z 223.237,A -85,B 0,C 180,E1 -17474.674,E2 -17474.674} C_VEL
LIN {X 0,Y 277.344,Z 223.222,A -85,B 0,C 180,E1 -17479.234,E2 -17479.234} C_VEL
LIN {X 0,Y 277.319,Z 223.236,A -85,B 0,C 180,E1 -17484.17,E2 -17484.17} C_VEL
LIN {X 0,Y 277.336,Z 223.243,A -85,B 0,C 180,E1 -17487.51,E2 -17487.51} C_VEL
LIN {X 0,Y 277.271,Z 223.248,A -85,B 0,C 180,E1 -17490.481,E2 -17490.481} C_VEL
LIN {X 0,Y 277.246,Z 223.254,A -85,B 0,C 180,E1 -17493.896,E2 -17493.896} C_VEL
LIN {X 0,Y 277.263,Z 223.24,A -85,B 0,C 180,E1 -17497.47,E2 -17497.47} C_VEL
LIN {X 0,Y 277.209,Z 223.269,A -85,B 0,C 180,E1 -17501.236,E2 -17501.236} C_VEL
LIN {X 0,Y 277.2,Z 223.259,A -85,B 0,C 180,E1 -17505.226,E2 -17505.226} C_VEL
LIN {X 0,Y 277.221,Z 223.249,A -85,B 0,C 180,E1 -17509.512,E2 -17509.512} C_VEL
LIN {X 0,Y 277.267,Z 223.251,A -85,B 0,C 180,E1 -17512.531,E2 -17512.531} C_VEL
LIN {X 0,Y 277.247,Z 223.265,A -85,B 0,C 180,E1 -17516.104,E2 -17516.104} C_VEL
LIN {X 0,Y 277.261,Z 223.25,A -85,B 0,C 180,E1 -17519.539,E2 -17519.539} C_VEL
LIN {X 0,Y 277.364,Z 223.281,A -85,B 0,C 180,E1 -17523.437,E2 -17523.437} C_VEL
LIN {X 0,Y 278.201,Z 225.875,A -85,B 0,C 180,E1 -17523.734,E2 -17523.734} C_VEL
LIN {X 0,Y 280.074,Z 228.022,A -85,B 0,C 180,E1 -17524.242,E2 -17524.242} C_VEL
LIN {X 0,Y 280.784,Z 228.953,A -85,B 0,C 180,E1 -17524.438,E2 -17524.438} C_VEL
LIN {X 0,Y 282.957,Z 232.202,A -85,B 0,C 180,E1 -17525.042,E2 -17525.042} C_VEL
LIN {X 0,Y 284.145,Z 233.703,A -85,B 0,C 180,E1 -17525.355,E2 -17525.355} C_VEL
LIN {X 0,Y 293.37,Z 246.86,A -85,B 0,C 180,E1 -17527.703,E2 -17527.703} C_VEL
LIN {X 0,Y 300.772,Z 258.164,A -85,B 0,C 180,E1 -17529.469,E2 -17529.469} C_VEL
LIN {X 0,Y 310.032,Z 273.33,A -85,B 0,C 180,E1 -17531.54,E2 -17531.54} C_VEL
LIN {X 0,Y 316.227,Z 284.608,A -85,B 0,C 180,E1 -17532.872,E2 -17532.872} C_VEL
LIN {X 0,Y 318.442,Z 289.064,A -85,B 0,C 180,E1 -17533.345,E2 -17533.345} C_VEL
LIN {X 0,Y 311.987,Z 419.813,A -85,B 0,C 180,E1 -17536.374,E2 -17536.374} C_VEL
LIN {X 0,Y 310.427,Z 436.74,A -85,B 0,C 180,E1 -17536.998,E2 -17536.998} C_VEL
LIN {X 0,Y 308.376,Z 452.792,A -85,B 0,C 180,E1 -17537.83,E2 -17537.83} C_VEL
LIN {X 0,Y 305.87,Z 468.57,A -85,B 0,C 180,E1 -17538.905,E2 -17538.905} C_VEL
LIN {X 0,Y 303.21,Z 483.112,A -85,B 0,C 180,E1 -17540.157,E2 -17540.157} C_VEL
LIN {X 0,Y 299.935,Z 498.155,A -85,B 0,C 180,E1 -17541.748,E2 -17541.748} C_VEL
LIN {X 0,Y 296.24,Z 513.118,A -85,B 0,C 180,E1 -17543.7,E2 -17543.7} C_VEL
LIN {X 0,Y 293.119,Z 524.702,A -85,B 0,C 180,E1 -17545.53,E2 -17545.53} C_VEL
LIN {X 0,Y 289.565,Z 537.35,A -85,B 0,C 180,E1 -17547.913,E2 -17547.913} C_VEL
LIN {X 0,Y 286.422,Z 548.128,A -85,B 0,C 180,E1 -17550.351,E2 -17550.351} C_VEL
LIN {X 0,Y 283.303,Z 558.562,A -85,B 0,C 180,E1 -17553.199,E2 -17553.199} C_VEL
LIN {X 0,Y 280.796,Z 567.257,A -85,B 0,C 180,E1 -17556.106,E2 -17556.106} C_VEL
LIN {X 0,Y 278.996,Z 573.656,A -85,B 0,C 180,E1 -17558.693,E2 -17558.693} C_VEL
LIN {X 0,Y 277.432,Z 579.808,A -85,B 0,C 180,E1 -17561.692,E2 -17561.692} C_VEL
LIN {X 0,Y 276.286,Z 584.846,A -85,B 0,C 180,E1 -17564.846,E2 -17564.846} C_VEL
LIN {X 0,Y 275.508,Z 588.448,A -85,B 0,C 180,E1 -17567.824,E2 -17567.824} C_VEL
LIN {X 0,Y 275.082,Z 591.147,A -85,B 0,C 180,E1 -17570.957,E2 -17570.957} C_VEL
LIN {X 0,Y 274.854,Z 592.66,A -85,B 0,C 180,E1 -17574.149,E2 -17574.149} C_VEL
LIN {X 0,Y 274.862,Z 593.083,A -85,B 0,C 180,E1 -17577.402,E2 -17577.402} C_VEL
LIN {X 0,Y 275.108,Z 592.341,A -85,B 0,C 180,E1 -17580.725,E2 -17580.725} C_VEL
LIN {X 0,Y 275.639,Z 590.248,A -85,B 0,C 180,E1 -17584.12,E2 -17584.12} C_VEL
LIN {X 0,Y 276.579,Z 586.782,A -85,B 0,C 180,E1 -17587.578,E2 -17587.578} C_VEL
LIN {X 0,Y 278.052,Z 581.803,A -85,B 0,C 180,E1 -17591.083,E2 -17591.083} C_VEL
LIN {X 0,Y 279.637,Z 576.865,A -85,B 0,C 180,E1 -17593.8,E2 -17593.8} C_VEL
LIN {X 0,Y 281.56,Z 571.097,A -85,B 0,C 180,E1 -17596.373,E2 -17596.373} C_VEL
LIN {X 0,Y 284.027,Z 564.118,A -85,B 0,C 180,E1 -17598.997,E2 -17598.997} C_VEL
LIN {X 0,Y 287.589,Z 554.301,A -85,B 0,C 180,E1 -17602.004,E2 -17602.004} C_VEL
LIN {X 0,Y 291.36,Z 543.813,A -85,B 0,C 180,E1 -17604.626,E2 -17604.626} C_VEL
LIN {X 0,Y 295.242,Z 532.48,A -85,B 0,C 180,E1 -17606.98,E2 -17606.98} C_VEL
LIN {X 0,Y 299.27,Z 520.19,A -85,B 0,C 180,E1 -17609.096,E2 -17609.096} C_VEL
LIN {X 0,Y 303.334,Z 506.562,A -85,B 0,C 180,E1 -17611.046,E2 -17611.046} C_VEL
LIN {X 0,Y 307.338,Z 491.65,A -85,B 0,C 180,E1 -17612.784,E2 -17612.784} C_VEL
LIN {X 0,Y 310.609,Z 477.85,A -85,B 0,C 180,E1 -17614.077,E2 -17614.077} C_VEL
LIN {X 0,Y 313.171,Z 465.007,A -85,B 0,C 180,E1 -17615.092,E2 -17615.092} C_VEL
LIN {X 0,Y 313.704,Z 459.627,A -85,B 0,C 180,E1 -17615.537,E2 -17615.537} C_VEL
LIN {X 0,Y 312.245,Z 443.177,A -85,B 0,C 180,E1 -17617.201,E2 -17617.201} C_VEL
LIN {X 0,Y 312.518,Z 436.682,A -85,B 0,C 180,E1 -17617.601,E2 -17617.601} C_VEL
LIN {X 0,Y 314.286,Z 420.616,A -85,B 0,C 180,E1 -17618.163,E2 -17618.163} C_VEL
LIN {X 0,Y 321.731,Z 296.547,A -85,B 0,C 180,E1 -17621.104,E2 -17621.104} C_VEL
LIN {X 0,Y 316.98,Z 287.208,A -85,B 0,C 180,E1 -17622.498,E2 -17622.498} C_VEL
LIN {X 0,Y 310.562,Z 276.437,A -85,B 0,C 180,E1 -17624.473,E2 -17624.473} C_VEL
LIN {X 0,Y 304.629,Z 267.493,A -85,B 0,C 180,E1 -17626.458,E2 -17626.458} C_VEL
LIN {X 0,Y 299.26,Z 259.666,A -85,B 0,C 180,E1 -17628.459,E2 -17628.459} C_VEL
LIN {X 0,Y 296.199,Z 255.613,A -85,B 0,C 180,E1 -17629.68,E2 -17629.68} C_VEL
LIN {X 0,Y 292.736,Z 251.059,A -85,B 0,C 180,E1 -17631.168,E2 -17631.168} C_VEL
LIN {X 0,Y 289.869,Z 247.28,A -85,B 0,C 180,E1 -17632.532,E2 -17632.532} C_VEL
LIN {X 0,Y 288.717,Z 245.951,A -85,B 0,C 180,E1 -17633.096,E2 -17633.096} C_VEL
LIN {X 0,Y 286.119,Z 242.7,A -85,B 0,C 180,E1 -17634.45,E2 -17634.45} C_VEL
LIN {X 0,Y 285.377,Z 241.482,A -85,B 0,C 180,E1 -17634.878,E2 -17634.878} C_VEL
LIN {X 0,Y 282.523,Z 239.023,A -85,B 0,C 180,E1 -17636.524,E2 -17636.524} C_VEL
LIN {X 0,Y 280.921,Z 236.034,A -85,B 0,C 180,E1 -17637.661,E2 -17637.661} C_VEL
LIN {X 0,Y 277.874,Z 233.443,A -85,B 0,C 180,E1 -17639.819,E2 -17639.819} C_VEL
LIN {X 0,Y 276.361,Z 230.448,A -85,B 0,C 180,E1 -17641.275,E2 -17641.275} C_VEL
LIN {X 0,Y 276.181,Z 230.099,A -85,B 0,C 180,E1 -17641.458,E2 -17641.458} C_VEL
LIN {X 0,Y 272.741,Z 228.515,A -85,B 0,C 180,E1 -17644.989,E2 -17644.989} C_VEL
LIN {X 0,Y 270.55,Z 224.606,A -85,B 0,C 180,E1 -17649.72,E2 -17649.72} C_VEL
LIN {X 0,Y 270.377,Z 224.112,A -85,B 0,C 180,E1 -17650.862,E2 -17650.862} C_VEL
LIN {X 0,Y 270.409,Z 224.221,A -85,B 0,C 180,E1 -17655.219,E2 -17655.219} C_VEL
LIN {X 0,Y 272.134,Z 228.069,A -85,B 0,C 180,E1 -17659.78,E2 -17659.78} C_VEL
LIN {X 0,Y 274.783,Z 229.9,A -85,B 0,C 180,E1 -17662.966,E2 -17662.966} C_VEL
LIN {X 0,Y 275.838,Z 230.375,A -85,B 0,C 180,E1 -17663.925,E2 -17663.925} C_VEL
LIN {X 0,Y 276.918,Z 232.913,A -85,B 0,C 180,E1 -17665.057,E2 -17665.057} C_VEL
LIN {X 0,Y 279.544,Z 235.443,A -85,B 0,C 180,E1 -17667.1,E2 -17667.1} C_VEL
LIN {X 0,Y 280.796,Z 236.283,A -85,B 0,C 180,E1 -17667.919,E2 -17667.919} C_VEL
LIN {X 0,Y 282.698,Z 239.494,A -85,B 0,C 180,E1 -17669.24,E2 -17669.24} C_VEL
LIN {X 0,Y 285.286,Z 242.011,A -85,B 0,C 180,E1 -17670.75,E2 -17670.75} C_VEL
LIN {X 0,Y 291.278,Z 250.045,A -85,B 0,C 180,E1 -17673.837,E2 -17673.837} C_VEL
LIN {X 0,Y 295.368,Z 255.95,A -85,B 0,C 180,E1 -17675.685,E2 -17675.685} C_VEL
LIN {X 0,Y 299.91,Z 262.805,A -85,B 0,C 180,E1 -17677.537,E2 -17677.537} C_VEL
LIN {X 0,Y 305.737,Z 272.366,A -85,B 0,C 180,E1 -17679.704,E2 -17679.704} C_VEL
LIN {X 0,Y 312.083,Z 283.548,A -85,B 0,C 180,E1 -17681.836,E2 -17681.836} C_VEL
LIN {X 0,Y 318.006,Z 295.37,A -85,B 0,C 180,E1 -17683.68,E2 -17683.68} C_VEL
LIN {X 0,Y 321.518,Z 303.177,A -85,B 0,C 180,E1 -17684.725,E2 -17684.725} C_VEL
LIN {X 0,Y 313.643,Z 433.464,A -85,B 0,C 180,E1 -17687.797,E2 -17687.797} C_VEL
LIN {X 0,Y 311.662,Z 450.266,A -85,B 0,C 180,E1 -17688.386,E2 -17688.386} C_VEL
LIN {X 0,Y 309.067,Z 466.342,A -85,B 0,C 180,E1 -17689.176,E2 -17689.176} C_VEL
LIN {X 0,Y 305.962,Z 481.953,A -85,B 0,C 180,E1 -17690.188,E2 -17690.188} C_VEL
LIN {X 0,Y 302.653,Z 496.453,A -85,B 0,C 180,E1 -17691.387,E2 -17691.387} C_VEL
LIN {X 0,Y 298.625,Z 511.352,A -85,B 0,C 180,E1 -17692.911,E2 -17692.911} C_VEL
LIN {X 0,Y 294.457,Z 525.307,A -85,B 0,C 180,E1 -17694.68,E2 -17694.68} C_VEL
LIN {X 0,Y 290.343,Z 537.817,A -85,B 0,C 180,E1 -17696.587,E2 -17696.587} C_VEL
LIN {X 0,Y 285.971,Z 550.501,A -85,B 0,C 180,E1 -17698.93,E2 -17698.93} C_VEL
LIN {X 0,Y 282.16,Z 561.353,A -85,B 0,C 180,E1 -17701.35,E2 -17701.35} C_VEL
LIN {X 0,Y 278.331,Z 571.822,A -85,B 0,C 180,E1 -17704.179,E2 -17704.179} C_VEL
LIN {X 0,Y 275.298,Z 580.246,A -85,B 0,C 180,E1 -17706.935,E2 -17706.935} C_VEL
LIN {X 0,Y 272.964,Z 587.242,A -85,B 0,C 180,E1 -17709.661,E2 -17709.661} C_VEL
LIN {X 0,Y 270.555,Z 594.915,A -85,B 0,C 180,E1 -17713.398,E2 -17713.398} C_VEL
LIN {X 0,Y 269.1,Z 600.794,A -85,B 0,C 180,E1 -17717.175,E2 -17717.175} C_VEL
LIN {X 0,Y 268.308,Z 604.994,A -85,B 0,C 180,E1 -17720.958,E2 -17720.958} C_VEL
LIN {X 0,Y 268.129,Z 607.691,A -85,B 0,C 180,E1 -17724.889,E2 -17724.889} C_VEL
LIN {X 0,Y 268.146,Z 608.465,A -85,B 0,C 180,E1 -17726.996,E2 -17726.996} C_VEL
LIN {X 0,Y 268.2,Z 608.688,A -85,B 0,C 180,E1 -17730,E2 -17730} C_VEL
LIN {X 0,Y 268.155,Z 607.995,A -85,B 0,C 180,E1 -17733.005,E2 -17733.005} C_VEL
LIN {X 0,Y 268.138,Z 606.22,A -85,B 0,C 180,E1 -17736.018,E2 -17736.018} C_VEL
LIN {X 0,Y 268.304,Z 603.505,A -85,B 0,C 180,E1 -17739.043,E2 -17739.043} C_VEL
LIN {X 0,Y 269.04,Z 598.537,A -85,B 0,C 180,E1 -17742.829,E2 -17742.829} C_VEL
LIN {X 0,Y 270.055,Z 593.612,A -85,B 0,C 180,E1 -17745.657,E2 -17745.657} C_VEL
LIN {X 0,Y 271.662,Z 586.739,A -85,B 0,C 180,E1 -17748.868,E2 -17748.868} C_VEL
LIN {X 0,Y 273.828,Z 578.885,A -85,B 0,C 180,E1 -17751.849,E2 -17751.849} C_VEL
LIN {X 0,Y 276.578,Z 569.395,A -85,B 0,C 180,E1 -17754.789,E2 -17754.789} C_VEL
LIN {X 0,Y 279.584,Z 559.606,A -85,B 0,C 180,E1 -17757.307,E2 -17757.307} C_VEL
LIN {X 0,Y 282.621,Z 549.186,A -85,B 0,C 180,E1 -17759.591,E2 -17759.591} C_VEL
LIN {X 0,Y 286.245,Z 536.717,A -85,B 0,C 180,E1 -17761.862,E2 -17761.862} C_VEL
LIN {X 0,Y 289.655,Z 524.439,A -85,B 0,C 180,E1 -17763.712,E2 -17763.712} C_VEL
LIN {X 0,Y 293.307,Z 510.315,A -85,B 0,C 180,E1 -17765.483,E2 -17765.483} C_VEL
LIN {X 0,Y 296.602,Z 495.979,A -85,B 0,C 180,E1 -17766.96,E2 -17766.96} C_VEL
LIN {X 0,Y 299.634,Z 480.855,A -85,B 0,C 180,E1 -17768.216,E2 -17768.216} C_VEL
LIN {X 0,Y 302.176,Z 465.42,A -85,B 0,C 180,E1 -17769.222,E2 -17769.222} C_VEL
LIN {X 0,Y 304.369,Z 449.259,A -85,B 0,C 180,E1 -17770.01,E2 -17770.01} C_VEL
LIN {X 0,Y 306.076,Z 432.828,A -85,B 0,C 180,E1 -17770.561,E2 -17770.561} C_VEL
LIN {X 0,Y 312.824,Z 299.242,A -85,B 0,C 180,E1 -17773.702,E2 -17773.702} C_VEL
LIN {X 0,Y 303.233,Z 279.503,A -85,B 0,C 180,E1 -17775.891,E2 -17775.891} C_VEL
LIN {X 0,Y 295.013,Z 264.347,A -85,B 0,C 180,E1 -17777.875,E2 -17777.875} C_VEL
LIN {X 0,Y 284.93,Z 247.302,A -85,B 0,C 180,E1 -17780.477,E2 -17780.477} C_VEL
LIN {X 0,Y 277.422,Z 235.781,A -85,B 0,C 180,E1 -17782.555,E2 -17782.555} C_VEL
LIN {X 0,Y 273.514,Z 229.951,A -85,B 0,C 180,E1 -17783.703,E2 -17783.703} C_VEL
LIN {X 0,Y 270.791,Z 226.144,A -85,B 0,C 180,E1 -17784.525,E2 -17784.525} C_VEL
LIN {X 0,Y 270.194,Z 224.133,A -85,B 0,C 180,E1 -17785.18,E2 -17785.18} C_VEL
LIN {X 0,Y 270.199,Z 224.117,A -85,B 0,C 180,E1 -17789.131,E2 -17789.131} C_VEL
LIN {X 0,Y 270.263,Z 224.121,A -85,B 0,C 180,E1 -17792.146,E2 -17792.146} C_VEL
LIN {X 0,Y 270.276,Z 224.11,A -85,B 0,C 180,E1 -17795.519,E2 -17795.519} C_VEL
LIN {X 0,Y 270.269,Z 224.095,A -85,B 0,C 180,E1 -17800.242,E2 -17800.242} C_VEL
LIN {X 0,Y 270.376,Z 224.116,A -85,B 0,C 180,E1 -17804.934,E2 -17804.934} C_VEL
LIN {X 0,Y 270.387,Z 224.078,A -85,B 0,C 180,E1 -17809.517,E2 -17809.517} C_VEL
LIN {X 0,Y 270.583,Z 224.094,A -85,B 0,C 180,E1 -17812.538,E2 -17812.538} C_VEL
LIN {X 0,Y 270.784,Z 224.024,A -85,B 0,C 180,E1 -17818.513,E2 -17818.513} C_VEL
LIN {X 0,Y 270.785,Z 224.067,A -85,B 0,C 180,E1 -17821.487,E2 -17821.487} C_VEL
LIN {X 0,Y 270.598,Z 224.085,A -85,B 0,C 180,E1 -17827.462,E2 -17827.462} C_VEL
LIN {X 0,Y 270.412,Z 224.095,A -85,B 0,C 180,E1 -17830.482,E2 -17830.482} C_VEL
LIN {X 0,Y 270.402,Z 224.113,A -85,B 0,C 180,E1 -17835.065,E2 -17835.065} C_VEL
LIN {X 0,Y 270.301,Z 224.102,A -85,B 0,C 180,E1 -17839.756,E2 -17839.756} C_VEL
LIN {X 0,Y 270.274,Z 224.108,A -85,B 0,C 180,E1 -17844.586,E2 -17844.586} C_VEL
LIN {X 0,Y 270.275,Z 224.126,A -85,B 0,C 180,E1 -17847.908,E2 -17847.908} C_VEL
LIN {X 0,Y 270.184,Z 224.12,A -85,B 0,C 180,E1 -17851.348,E2 -17851.348} C_VEL
LIN {X 0,Y 270.201,Z 224.14,A -85,B 0,C 180,E1 -17854.905,E2 -17854.905} C_VEL
LIN {X 0,Y 270.197,Z 224.119,A -85,B 0,C 180,E1 -17858.71,E2 -17858.71} C_VEL
LIN {X 0,Y 270.171,Z 224.132,A -85,B 0,C 180,E1 -17862.558,E2 -17862.558} C_VEL
LIN {X 0,Y 270.164,Z 224.146,A -85,B 0,C 180,E1 -17866.751,E2 -17866.751} C_VEL
LIN {X 0,Y 270.173,Z 224.127,A -85,B 0,C 180,E1 -17869.434,E2 -17869.434} C_VEL
LIN {X 0,Y 270.225,Z 224.118,A -85,B 0,C 180,E1 -17873.73,E2 -17873.73} C_VEL
LIN {X 0,Y 270.202,Z 224.139,A -85,B 0,C 180,E1 -17876.892,E2 -17876.892} C_VEL
LIN {X 0,Y 270.253,Z 224.131,A -85,B 0,C 180,E1 -17881.328,E2 -17881.328} C_VEL
LIN {X 0,Y 270.255,Z 224.125,A -85,B 0,C 180,E1 -17881.773,E2 -17881.773} C_VEL
LIN {X 0,Y 271.158,Z 226.802,A -85,B 0,C 180,E1 -17882.115,E2 -17882.115} C_VEL
LIN {X 0,Y 273.26,Z 229.036,A -85,B 0,C 180,E1 -17882.716,E2 -17882.716} C_VEL
LIN {X 0,Y 273.892,Z 229.888,A -85,B 0,C 180,E1 -17882.901,E2 -17882.901} C_VEL
LIN {X 0,Y 275.949,Z 233.051,A -85,B 0,C 180,E1 -17883.509,E2 -17883.509} C_VEL
LIN {X 0,Y 277.447,Z 234.935,A -85,B 0,C 180,E1 -17883.928,E2 -17883.928} C_VEL
LIN {X 0,Y 286.564,Z 247.797,A -85,B 0,C 180,E1 -17886.391,E2 -17886.391} C_VEL
LIN {X 0,Y 294.483,Z 259.659,A -85,B 0,C 180,E1 -17888.368,E2 -17888.368} C_VEL
LIN {X 0,Y 304.504,Z 275.947,A -85,B 0,C 180,E1 -17890.712,E2 -17890.712} C_VEL
LIN {X 0,Y 311.538,Z 288.811,A -85,B 0,C 180,E1 -17892.272,E2 -17892.272} C_VEL
LIN {X 0,Y 312.865,Z 291.501,A -85,B 0,C 180,E1 -17892.565,E2 -17892.565} C_VEL
LIN {X 0,Y 306.307,Z 419.991,A -85,B 0,C 180,E1 -17895.585,E2 -17895.585} C_VEL
LIN {X 0,Y 304.731,Z 436.656,A -85,B 0,C 180,E1 -17896.206,E2 -17896.206} C_VEL
LIN {X 0,Y 302.698,Z 452.295,A -85,B 0,C 180,E1 -17897.02,E2 -17897.02} C_VEL
LIN {X 0,Y 300.176,Z 467.989,A -85,B 0,C 180,E1 -17898.093,E2 -17898.093} C_VEL
LIN {X 0,Y 297.202,Z 483.513,A -85,B 0,C 180,E1 -17899.44,E2 -17899.44} C_VEL
LIN {X 0,Y 293.807,Z 498.544,A -85,B 0,C 180,E1 -17901.055,E2 -17901.055} C_VEL
LIN {X 0,Y 290.012,Z 513.468,A -85,B 0,C 180,E1 -17903.04,E2 -17903.04} C_VEL
LIN {X 0,Y 286.508,Z 526.013,A -85,B 0,C 180,E1 -17905.074,E2 -17905.074} C_VEL
LIN {X 0,Y 282.85,Z 538.483,A -85,B 0,C 180,E1 -17907.507,E2 -17907.507} C_VEL
LIN {X 0,Y 279.604,Z 549.114,A -85,B 0,C 180,E1 -17910,E2 -17910} C_VEL
LIN {X 0,Y 276.767,Z 558.262,A -85,B 0,C 180,E1 -17912.546,E2 -17912.546} C_VEL
LIN {X 0,Y 274.147,Z 566.922,A -85,B 0,C 180,E1 -17915.479,E2 -17915.479} C_VEL
LIN {X 0,Y 272.201,Z 573.517,A -85,B 0,C 180,E1 -17918.163,E2 -17918.163} C_VEL
LIN {X 0,Y 270.541,Z 579.737,A -85,B 0,C 180,E1 -17921.234,E2 -17921.234} C_VEL
LIN {X 0,Y 269.103,Z 585.762,A -85,B 0,C 180,E1 -17925.138,E2 -17925.138} C_VEL
LIN {X 0,Y 268.351,Z 589.272,A -85,B 0,C 180,E1 -17928.316,E2 -17928.316} C_VEL
LIN {X 0,Y 267.915,Z 591.713,A -85,B 0,C 180,E1 -17931.545,E2 -17931.545} C_VEL
LIN {X 0,Y 267.732,Z 593.085,A -85,B 0,C 180,E1 -17934.834,E2 -17934.834} C_VEL
LIN {X 0,Y 267.798,Z 593.229,A -85,B 0,C 180,E1 -17938.188,E2 -17938.188} C_VEL
LIN {X 0,Y 268.109,Z 592.202,A -85,B 0,C 180,E1 -17941.618,E2 -17941.618} C_VEL
LIN {X 0,Y 268.783,Z 589.901,A -85,B 0,C 180,E1 -17945.116,E2 -17945.116} C_VEL
LIN {X 0,Y 269.891,Z 586.16,A -85,B 0,C 180,E1 -17948.678,E2 -17948.678} C_VEL
LIN {X 0,Y 271.591,Z 580.831,A -85,B 0,C 180,E1 -17952.283,E2 -17952.283} C_VEL
LIN {X 0,Y 273.324,Z 575.712,A -85,B 0,C 180,E1 -17954.999,E2 -17954.999} C_VEL
LIN {X 0,Y 276.081,Z 568.406,A -85,B 0,C 180,E1 -17958.154,E2 -17958.154} C_VEL
LIN {X 0,Y 279.416,Z 559.536,A -85,B 0,C 180,E1 -17961.234,E2 -17961.234} C_VEL
LIN {X 0,Y 283.019,Z 550.047,A -85,B 0,C 180,E1 -17963.915,E2 -17963.915} C_VEL
LIN {X 0,Y 286.949,Z 539.548,A -85,B 0,C 180,E1 -17966.379,E2 -17966.379} C_VEL
LIN {X 0,Y 290.99,Z 527.847,A -85,B 0,C 180,E1 -17968.689,E2 -17968.689} C_VEL
LIN {X 0,Y 295.029,Z 515.833,A -85,B 0,C 180,E1 -17970.639,E2 -17970.639} C_VEL
LIN {X 0,Y 298.961,Z 502.661,A -85,B 0,C 180,E1 -17972.422,E2 -17972.422} C_VEL
LIN {X 0,Y 302.803,Z 488.313,A -85,B 0,C 180,E1 -17974.022,E2 -17974.022} C_VEL
LIN {X 0,Y 306.278,Z 473.728,A -85,B 0,C 180,E1 -17975.335,E2 -17975.335} C_VEL
LIN {X 0,Y 309.156,Z 459.07,A -85,B 0,C 180,E1 -17976.405,E2 -17976.405} C_VEL
LIN {X 0,Y 311.616,Z 443.453,A -85,B 0,C 180,E1 -17977.291,E2 -17977.291} C_VEL
LIN {X 0,Y 312.518,Z 436.682,A -85,B 0,C 180,E1 -17977.601,E2 -17977.601} C_VEL
LIN {X 0,Y 312.825,Z 431.009,A -85,B 0,C 180,E1 -17977.91,E2 -17977.91} C_VEL
LIN {X 0,Y 310.52,Z 413.647,A -85,B 0,C 180,E1 -17979.196,E2 -17979.196} C_VEL
LIN {X 0,Y 310.294,Z 408.877,A -85,B 0,C 180,E1 -17979.416,E2 -17979.416} C_VEL
LIN {X 0,Y 310.383,Z 406.931,A -85,B 0,C 180,E1 -17979.468,E2 -17979.468} C_VEL
LIN {X 0,Y 317.108,Z 299.602,A -85,B 0,C 180,E1 -17981.997,E2 -17981.997} C_VEL
LIN {X 0,Y 312.884,Z 291.241,A -85,B 0,C 180,E1 -17983.298,E2 -17983.298} C_VEL
LIN {X 0,Y 306.042,Z 279.776,A -85,B 0,C 180,E1 -17985.522,E2 -17985.522} C_VEL
LIN {X 0,Y 299.404,Z 269.666,A -85,B 0,C 180,E1 -17987.92,E2 -17987.92} C_VEL
LIN {X 0,Y 294.234,Z 262.234,A -85,B 0,C 180,E1 -17990.01,E2 -17990.01} C_VEL
LIN {X 0,Y 290.354,Z 257.177,A -85,B 0,C 180,E1 -17991.74,E2 -17991.74} C_VEL
LIN {X 0,Y 287.016,Z 252.657,A -85,B 0,C 180,E1 -17993.401,E2 -17993.401} C_VEL
LIN {X 0,Y 284.281,Z 249.339,A -85,B 0,C 180,E1 -17994.858,E2 -17994.858} C_VEL
LIN {X 0,Y 283.424,Z 248.001,A -85,B 0,C 180,E1 -17995.378,E2 -17995.378} C_VEL
LIN {X 0,Y 280.672,Z 245.409,A -85,B 0,C 180,E1 -17997.04,E2 -17997.04} C_VEL
LIN {X 0,Y 279.057,Z 242.539,A -85,B 0,C 180,E1 -17998.215,E2 -17998.215} C_VEL
LIN {X 0,Y 276.329,Z 240.024,A -85,B 0,C 180,E1 -18000.273,E2 -18000.273} C_VEL
LIN {X 0,Y 274.765,Z 237.005,A -85,B 0,C 180,E1 -18001.832,E2 -18001.832} C_VEL
LIN {X 0,Y 271.625,Z 235.456,A -85,B 0,C 180,E1 -18005.196,E2 -18005.196} C_VEL
LIN {X 0,Y 269.502,Z 231.449,A -85,B 0,C 180,E1 -18010.138,E2 -18010.138} C_VEL
LIN {X 0,Y 269.178,Z 231.109,A -85,B 0,C 180,E1 -18012.056,E2 -18012.056} C_VEL
LIN {X 0,Y 269.472,Z 231.48,A -85,B 0,C 180,E1 -18015.398,E2 -18015.398} C_VEL
LIN {X 0,Y 270.994,Z 234.959,A -85,B 0,C 180,E1 -18019.506,E2 -18019.506} C_VEL
LIN {X 0,Y 273.893,Z 236.967,A -85,B 0,C 180,E1 -18023.045,E2 -18023.045} C_VEL
LIN {X 0,Y 274.458,Z 237.398,A -85,B 0,C 180,E1 -18023.586,E2 -18023.586} C_VEL
LIN {X 0,Y 275.935,Z 240.264,A -85,B 0,C 180,E1 -18025.089,E2 -18025.089} C_VEL
LIN {X 0,Y 279.166,Z 243.104,A -85,B 0,C 180,E1 -18027.53,E2 -18027.53} C_VEL
LIN {X 0,Y 281.417,Z 246.57,A -85,B 0,C 180,E1 -18029.096,E2 -18029.096} C_VEL
LIN {X 0,Y 283.602,Z 248.694,A -85,B 0,C 180,E1 -18030.396,E2 -18030.396} C_VEL
LIN {X 0,Y 289.107,Z 256.342,A -85,B 0,C 180,E1 -18033.34,E2 -18033.34} C_VEL
LIN {X 0,Y 292.882,Z 261.944,A -85,B 0,C 180,E1 -18035.123,E2 -18035.123} C_VEL
LIN {X 0,Y 297.029,Z 268.369,A -85,B 0,C 180,E1 -18036.887,E2 -18036.887} C_VEL
LIN {X 0,Y 302.684,Z 277.857,A -85,B 0,C 180,E1 -18039.09,E2 -18039.09} C_VEL
LIN {X 0,Y 308.726,Z 288.813,A -85,B 0,C 180,E1 -18041.208,E2 -18041.208} C_VEL
LIN {X 0,Y 314.255,Z 300.134,A -85,B 0,C 180,E1 -18043.008,E2 -18043.008} C_VEL
LIN {X 0,Y 316.805,Z 305.817,A -85,B 0,C 180,E1 -18043.806,E2 -18043.806} C_VEL
LIN {X 0,Y 308.789,Z 432.963,A -85,B 0,C 180,E1 -18046.827,E2 -18046.827} C_VEL
LIN {X 0,Y 306.764,Z 450.08,A -85,B 0,C 180,E1 -18047.437,E2 -18047.437} C_VEL
LIN {X 0,Y 304.033,Z 466.362,A -85,B 0,C 180,E1 -18048.24,E2 -18048.24} C_VEL
LIN {X 0,Y 300.59,Z 482.847,A -85,B 0,C 180,E1 -18049.329,E2 -18049.329} C_VEL
LIN {X 0,Y 296.748,Z 498.642,A -85,B 0,C 180,E1 -18050.69,E2 -18050.69} C_VEL
LIN {X 0,Y 292.889,Z 512.273,A -85,B 0,C 180,E1 -18052.123,E2 -18052.123} C_VEL
LIN {X 0,Y 288.665,Z 525.8,A -85,B 0,C 180,E1 -18053.879,E2 -18053.879} C_VEL
LIN {X 0,Y 284.424,Z 538.11,A -85,B 0,C 180,E1 -18055.797,E2 -18055.797} C_VEL
LIN {X 0,Y 280.499,Z 549.078,A -85,B 0,C 180,E1 -18057.832,E2 -18057.832} C_VEL
LIN {X 0,Y 276.45,Z 560.007,A -85,B 0,C 180,E1 -18060.283,E2 -18060.283} C_VEL
LIN {X 0,Y 272.792,Z 569.412,A -85,B 0,C 180,E1 -18062.788,E2 -18062.788} C_VEL
LIN {X 0,Y 269.695,Z 577.588,A -85,B 0,C 180,E1 -18065.359,E2 -18065.359} C_VEL
LIN {X 0,Y 266.843,Z 585.424,A -85,B 0,C 180,E1 -18068.364,E2 -18068.364} C_VEL
LIN {X 0,Y 264.582,Z 591.985,A -85,B 0,C 180,E1 -18071.413,E2 -18071.413} C_VEL
LIN {X 0,Y 262.953,Z 597.368,A -85,B 0,C 180,E1 -18074.499,E2 -18074.499} C_VEL
LIN {X 0,Y 261.873,Z 601.601,A -85,B 0,C 180,E1 -18077.603,E2 -18077.603} C_VEL
LIN {X 0,Y 261.235,Z 604.859,A -85,B 0,C 180,E1 -18080.711,E2 -18080.711} C_VEL
LIN {X 0,Y 261.034,Z 607.018,A -85,B 0,C 180,E1 -18083.818,E2 -18083.818} C_VEL
LIN {X 0,Y 261.04,Z 608.282,A -85,B 0,C 180,E1 -18086.914,E2 -18086.914} C_VEL
LIN {X 0,Y 261.126,Z 608.474,A -85,B 0,C 180,E1 -18090,E2 -18090} C_VEL
LIN {X 0,Y 261.069,Z 607.763,A -85,B 0,C 180,E1 -18093.087,E2 -18093.087} C_VEL
LIN {X 0,Y 261.035,Z 605.956,A -85,B 0,C 180,E1 -18096.183,E2 -18096.183} C_VEL
LIN {X 0,Y 261.231,Z 603.212,A -85,B 0,C 180,E1 -18099.29,E2 -18099.29} C_VEL
LIN {X 0,Y 262.041,Z 598.209,A -85,B 0,C 180,E1 -18103.178,E2 -18103.178} C_VEL
LIN {X 0,Y 263.199,Z 592.802,A -85,B 0,C 180,E1 -18106.318,E2 -18106.318} C_VEL
LIN {X 0,Y 264.851,Z 586.327,A -85,B 0,C 180,E1 -18109.372,E2 -18109.372} C_VEL
LIN {X 0,Y 267.139,Z 578.439,A -85,B 0,C 180,E1 -18112.425,E2 -18112.425} C_VEL
LIN {X 0,Y 270.03,Z 568.903,A -85,B 0,C 180,E1 -18115.432,E2 -18115.432} C_VEL
LIN {X 0,Y 273.197,Z 559.056,A -85,B 0,C 180,E1 -18118.001,E2 -18118.001} C_VEL
LIN {X 0,Y 276.668,Z 547.532,A -85,B 0,C 180,E1 -18120.534,E2 -18120.534} C_VEL
LIN {X 0,Y 280.486,Z 534.983,A -85,B 0,C 180,E1 -18122.809,E2 -18122.809} C_VEL
LIN {X 0,Y 284.384,Z 521.354,A -85,B 0,C 180,E1 -18124.845,E2 -18124.845} C_VEL
LIN {X 0,Y 288.233,Z 506.259,A -85,B 0,C 180,E1 -18126.682,E2 -18126.682} C_VEL
LIN {X 0,Y 291.719,Z 491.395,A -85,B 0,C 180,E1 -18128.123,E2 -18128.123} C_VEL
LIN {X 0,Y 294.598,Z 476.263,A -85,B 0,C 180,E1 -18129.322,E2 -18129.322} C_VEL
LIN {X 0,Y 297.247,Z 459.684,A -85,B 0,C 180,E1 -18130.334,E2 -18130.334} C_VEL
LIN {X 0,Y 299.359,Z 443.583,A -85,B 0,C 180,E1 -18131.042,E2 -18131.042} C_VEL
LIN {X 0,Y 300.784,Z 427.066,A -85,B 0,C 180,E1 -18131.533,E2 -18131.533} C_VEL
LIN {X 0,Y 307.263,Z 301.519,A -85,B 0,C 180,E1 -18134.507,E2 -18134.507} C_VEL
LIN {X 0,Y 297.832,Z 282.056,A -85,B 0,C 180,E1 -18136.748,E2 -18136.748} C_VEL
LIN {X 0,Y 289.158,Z 266.154,A -85,B 0,C 180,E1 -18138.925,E2 -18138.925} C_VEL
LIN {X 0,Y 280.845,Z 252.086,A -85,B 0,C 180,E1 -18141.158,E2 -18141.158} C_VEL
LIN {X 0,Y 273.764,Z 241.076,A -85,B 0,C 180,E1 -18143.182,E2 -18143.182} C_VEL
LIN {X 0,Y 269.26,Z 234.253,A -85,B 0,C 180,E1 -18144.554,E2 -18144.554} C_VEL
LIN {X 0,Y 267.138,Z 231.368,A -85,B 0,C 180,E1 -18145.211,E2 -18145.211} C_VEL
LIN {X 0,Y 266.027,Z 229.89,A -85,B 0,C 180,E1 -18145.561,E2 -18145.561} C_VEL
LIN {X 0,Y 263.954,Z 227.487,A -85,B 0,C 180,E1 -18146.213,E2 -18146.213} C_VEL
LIN {X 0,Y 263.201,Z 225.213,A -85,B 0,C 180,E1 -18146.583,E2 -18146.583} C_VEL
LIN {X 0,Y 263.131,Z 224.997,A -85,B 0,C 180,E1 -18147.712,E2 -18147.712} C_VEL
LIN {X 0,Y 263.199,Z 225.007,A -85,B 0,C 180,E1 -18151.784,E2 -18151.784} C_VEL
LIN {X 0,Y 263.225,Z 224.984,A -85,B 0,C 180,E1 -18155.201,E2 -18155.201} C_VEL
LIN {X 0,Y 263.25,Z 224.973,A -85,B 0,C 180,E1 -18159.692,E2 -18159.692} C_VEL
LIN {X 0,Y 263.322,Z 224.998,A -85,B 0,C 180,E1 -18164.52,E2 -18164.52} C_VEL
LIN {X 0,Y 263.333,Z 224.952,A -85,B 0,C 180,E1 -18169.233,E2 -18169.233} C_VEL
LIN {X 0,Y 263.543,Z 224.97,A -85,B 0,C 180,E1 -18172.338,E2 -18172.338} C_VEL
LIN {X 0,Y 263.748,Z 224.898,A -85,B 0,C 180,E1 -18178.473,E2 -18178.473} C_VEL
LIN {X 0,Y 263.75,Z 224.944,A -85,B 0,C 180,E1 -18181.527,E2 -18181.527} C_VEL
LIN {X 0,Y 263.557,Z 224.963,A -85,B 0,C 180,E1 -18187.662,E2 -18187.662} C_VEL
LIN {X 0,Y 263.354,Z 224.97,A -85,B 0,C 180,E1 -18190.766,E2 -18190.766} C_VEL
LIN {X 0,Y 263.35,Z 224.992,A -85,B 0,C 180,E1 -18195.478,E2 -18195.478} C_VEL
LIN {X 0,Y 263.263,Z 224.985,A -85,B 0,C 180,E1 -18200.307,E2 -18200.307} C_VEL
LIN {X 0,Y 263.209,Z 224.983,A -85,B 0,C 180,E1 -18205.291,E2 -18205.291} C_VEL
LIN {X 0,Y 263.183,Z 225.014,A -85,B 0,C 180,E1 -18208.729,E2 -18208.729} C_VEL
LIN {X 0,Y 263.132,Z 224.995,A -85,B 0,C 180,E1 -18212.288,E2 -18212.288} C_VEL
LIN {X 0,Y 263.181,Z 225.001,A -85,B 0,C 180,E1 -18216.763,E2 -18216.763} C_VEL
LIN {X 0,Y 263.124,Z 225.02,A -85,B 0,C 180,E1 -18221.593,E2 -18221.593} C_VEL
LIN {X 0,Y 263.123,Z 225.023,A -85,B 0,C 180,E1 -18226.151,E2 -18226.151} C_VEL
LIN {X 0,Y 263.105,Z 225.012,A -85,B 0,C 180,E1 -18230.127,E2 -18230.127} C_VEL
LIN {X 0,Y 263.162,Z 224.997,A -85,B 0,C 180,E1 -18234.018,E2 -18234.018} C_VEL
LIN {X 0,Y 263.133,Z 225.009,A -85,B 0,C 180,E1 -18237.712,E2 -18237.712} C_VEL
LIN {X 0,Y 263.16,Z 225.01,A -85,B 0,C 180,E1 -18239.981,E2 -18239.981} C_VEL
LIN {X 0,Y 263.984,Z 227.524,A -85,B 0,C 180,E1 -18240.314,E2 -18240.314} C_VEL
LIN {X 0,Y 265.876,Z 229.738,A -85,B 0,C 180,E1 -18240.909,E2 -18240.909} C_VEL
LIN {X 0,Y 266.807,Z 230.569,A -85,B 0,C 180,E1 -18241.186,E2 -18241.186} C_VEL
LIN {X 0,Y 268.842,Z 233.757,A -85,B 0,C 180,E1 -18241.84,E2 -18241.84} C_VEL
LIN {X 0,Y 270.511,Z 235.749,A -85,B 0,C 180,E1 -18242.336,E2 -18242.336} C_VEL
LIN {X 0,Y 274.58,Z 241.465,A -85,B 0,C 180,E1 -18243.536,E2 -18243.536} C_VEL
LIN {X 0,Y 282.697,Z 252.935,A -85,B 0,C 180,E1 -18245.783,E2 -18245.783} C_VEL
LIN {X 0,Y 290.494,Z 264.714,A -85,B 0,C 180,E1 -18247.792,E2 -18247.792} C_VEL
LIN {X 0,Y 300.831,Z 281.771,A -85,B 0,C 180,E1 -18250.276,E2 -18250.276} C_VEL
LIN {X 0,Y 307.27,Z 293.838,A -85,B 0,C 180,E1 -18251.751,E2 -18251.751} C_VEL
LIN {X 0,Y 305.604,Z 326.511,A -85,B 0,C 180,E1 -18252.529,E2 -18252.529} C_VEL
LIN {X 0,Y 300.607,Z 420.949,A -85,B 0,C 180,E1 -18254.794,E2 -18254.794} C_VEL
LIN {X 0,Y 298.908,Z 438.214,A -85,B 0,C 180,E1 -18255.46,E2 -18255.46} C_VEL
LIN {X 0,Y 296.596,Z 454.815,A -85,B 0,C 180,E1 -18256.364,E2 -18256.364} C_VEL
LIN {X 0,Y 293.936,Z 470.304,A -85,B 0,C 180,E1 -18257.477,E2 -18257.477} C_VEL
LIN {X 0,Y 290.92,Z 485.462,A -85,B 0,C 180,E1 -18258.856,E2 -18258.856} C_VEL
LIN {X 0,Y 287.749,Z 498.913,A -85,B 0,C 180,E1 -18260.333,E2 -18260.333} C_VEL
LIN {X 0,Y 284.071,Z 512.917,A -85,B 0,C 180,E1 -18262.223,E2 -18262.223} C_VEL
LIN {X 0,Y 280.467,Z 525.363,A -85,B 0,C 180,E1 -18264.247,E2 -18264.247} C_VEL
LIN {X 0,Y 276.646,Z 537.974,A -85,B 0,C 180,E1 -18266.723,E2 -18266.723} C_VEL
LIN {X 0,Y 273.217,Z 548.732,A -85,B 0,C 180,E1 -18269.263,E2 -18269.263} C_VEL
LIN {X 0,Y 269.88,Z 559.13,A -85,B 0,C 180,E1 -18272.238,E2 -18272.238} C_VEL
LIN {X 0,Y 267.154,Z 567.82,A -85,B 0,C 180,E1 -18275.282,E2 -18275.282} C_VEL
LIN {X 0,Y 264.924,Z 575.033,A -85,B 0,C 180,E1 -18278.389,E2 -18278.389} C_VEL
LIN {X 0,Y 263.269,Z 580.974,A -85,B 0,C 180,E1 -18281.549,E2 -18281.549} C_VEL
LIN {X 0,Y 262.015,Z 586.13,A -85,B 0,C 180,E1 -18285.067,E2 -18285.067} C_VEL
LIN {X 0,Y 261.167,Z 590.085,A -85,B 0,C 180,E1 -18288.839,E2 -18288.839} C_VEL
LIN {X 0,Y 260.785,Z 592.266,A -85,B 0,C 180,E1 -18292.165,E2 -18292.165} C_VEL
LIN {X 0,Y 260.613,Z 593.385,A -85,B 0,C 180,E1 -18295.56,E2 -18295.56} C_VEL
LIN {X 0,Y 260.745,Z 593.375,A -85,B 0,C 180,E1 -18299.022,E2 -18299.022} C_VEL
LIN {X 0,Y 261.143,Z 592.059,A -85,B 0,C 180,E1 -18302.563,E2 -18302.563} C_VEL
LIN {X 0,Y 262.031,Z 589.215,A -85,B 0,C 180,E1 -18306.425,E2 -18306.425} C_VEL
LIN {X 0,Y 263.251,Z 585.402,A -85,B 0,C 180,E1 -18309.845,E2 -18309.845} C_VEL
LIN {X 0,Y 264.685,Z 581.298,A -85,B 0,C 180,E1 -18312.644,E2 -18312.644} C_VEL
LIN {X 0,Y 267.124,Z 574.676,A -85,B 0,C 180,E1 -18316.188,E2 -18316.188} C_VEL
LIN {X 0,Y 270.126,Z 567.014,A -85,B 0,C 180,E1 -18319.426,E2 -18319.426} C_VEL
LIN {X 0,Y 273.382,Z 559.056,A -85,B 0,C 180,E1 -18322.176,E2 -18322.176} C_VEL
LIN {X 0,Y 277.143,Z 549.61,A -85,B 0,C 180,E1 -18324.865,E2 -18324.865} C_VEL
LIN {X 0,Y 281.45,Z 538.502,A -85,B 0,C 180,E1 -18327.479,E2 -18327.479} C_VEL
LIN {X 0,Y 285.708,Z 526.827,A -85,B 0,C 180,E1 -18329.754,E2 -18329.754} C_VEL
LIN {X 0,Y 290.074,Z 514.137,A -85,B 0,C 180,E1 -18331.798,E2 -18331.798} C_VEL
LIN {X 0,Y 294.013,Z 501.216,A -85,B 0,C 180,E1 -18333.531,E2 -18333.531} C_VEL
LIN {X 0,Y 298.036,Z 486.613,A -85,B 0,C 180,E1 -18335.129,E2 -18335.129} C_VEL
LIN {X 0,Y 301.667,Z 471.426,A -85,B 0,C 180,E1 -18336.467,E2 -18336.467} C_VEL
LIN {X 0,Y 304.662,Z 456.381,A -85,B 0,C 180,E1 -18337.525,E2 -18337.525} C_VEL
LIN {X 0,Y 307.171,Z 440.634,A -85,B 0,C 180,E1 -18338.381,E2 -18338.381} C_VEL
LIN {X 0,Y 309.161,Z 423.635,A -85,B 0,C 180,E1 -18339.031,E2 -18339.031} C_VEL
LIN {X 0,Y 310.383,Z 406.931,A -85,B 0,C 180,E1 -18339.468,E2 -18339.468} C_VEL
LIN {X 0,Y 310.365,Z 401.151,A -85,B 0,C 180,E1 -18339.682,E2 -18339.682} C_VEL
LIN {X 0,Y 307.718,Z 382.682,A -85,B 0,C 180,E1 -18340.935,E2 -18340.935} C_VEL
LIN {X 0,Y 307.609,Z 376.909,A -85,B 0,C 180,E1 -18341.178,E2 -18341.178} C_VEL
LIN {X 0,Y 312.428,Z 302.387,A -85,B 0,C 180,E1 -18342.966,E2 -18342.966} C_VEL
LIN {X 0,Y 308.375,Z 294.437,A -85,B 0,C 180,E1 -18344.283,E2 -18344.283} C_VEL
LIN {X 0,Y 301.753,Z 283.341,A -85,B 0,C 180,E1 -18346.564,E2 -18346.564} C_VEL
LIN {X 0,Y 295.742,Z 274.113,A -85,B 0,C 180,E1 -18348.877,E2 -18348.877} C_VEL
LIN {X 0,Y 291.394,Z 267.888,A -85,B 0,C 180,E1 -18350.728,E2 -18350.728} C_VEL
LIN {X 0,Y 288.113,Z 263.384,A -85,B 0,C 180,E1 -18352.271,E2 -18352.271} C_VEL
LIN {X 0,Y 284.865,Z 258.971,A -85,B 0,C 180,E1 -18353.941,E2 -18353.941} C_VEL
LIN {X 0,Y 282.121,Z 255.309,A -85,B 0,C 180,E1 -18355.504,E2 -18355.504} C_VEL
LIN {X 0,Y 280.817,Z 253.971,A -85,B 0,C 180,E1 -18356.286,E2 -18356.286} C_VEL
LIN {X 0,Y 278.442,Z 251.131,A -85,B 0,C 180,E1 -18357.853,E2 -18357.853} C_VEL
LIN {X 0,Y 277.291,Z 249.151,A -85,B 0,C 180,E1 -18358.729,E2 -18358.729} C_VEL
LIN {X 0,Y 274.649,Z 246.382,A -85,B 0,C 180,E1 -18360.875,E2 -18360.875} C_VEL
LIN {X 0,Y 273.375,Z 243.925,A -85,B 0,C 180,E1 -18362.196,E2 -18362.196} C_VEL
LIN {X 0,Y 270.389,Z 242.243,A -85,B 0,C 180,E1 -18365.594,E2 -18365.594} C_VEL
LIN {X 0,Y 268.502,Z 238.389,A -85,B 0,C 180,E1 -18370.367,E2 -18370.367} C_VEL
LIN {X 0,Y 268.317,Z 238.228,A -85,B 0,C 180,E1 -18374.277,E2 -18374.277} C_VEL
LIN {X 0,Y 268.496,Z 238.739,A -85,B 0,C 180,E1 -18375.424,E2 -18375.424} C_VEL
LIN {X 0,Y 270.289,Z 242.332,A -85,B 0,C 180,E1 -18379.921,E2 -18379.921} C_VEL
LIN {X 0,Y 273.073,Z 244.243,A -85,B 0,C 180,E1 -18383.21,E2 -18383.21} C_VEL
LIN {X 0,Y 274.682,Z 247.187,A -85,B 0,C 180,E1 -18384.87,E2 -18384.87} C_VEL
LIN {X 0,Y 277.596,Z 249.907,A -85,B 0,C 180,E1 -18387.163,E2 -18387.163} C_VEL
LIN {X 0,Y 280.014,Z 253.481,A -85,B 0,C 180,E1 -18388.87,E2 -18388.87} C_VEL
LIN {X 0,Y 281.812,Z 255.32,A -85,B 0,C 180,E1 -18389.973,E2 -18389.973} C_VEL
LIN {X 0,Y 286.786,Z 262.367,A -85,B 0,C 180,E1 -18392.746,E2 -18392.746} C_VEL
LIN {X 0,Y 290.661,Z 268.323,A -85,B 0,C 180,E1 -18394.659,E2 -18394.659} C_VEL
LIN {X 0,Y 294.503,Z 274.451,A -85,B 0,C 180,E1 -18396.358,E2 -18396.358} C_VEL
LIN {X 0,Y 299.747,Z 283.468,A -85,B 0,C 180,E1 -18398.48,E2 -18398.48} C_VEL
LIN {X 0,Y 305.404,Z 294.006,A -85,B 0,C 180,E1 -18400.556,E2 -18400.556} C_VEL
LIN {X 0,Y 310.632,Z 305.074,A -85,B 0,C 180,E1 -18402.347,E2 -18402.347} C_VEL
LIN {X 0,Y 312.168,Z 308.615,A -85,B 0,C 180,E1 -18402.852,E2 -18402.852} C_VEL
LIN {X 0,Y 303.978,Z 433.312,A -85,B 0,C 180,E1 -18405.855,E2 -18405.855} C_VEL
LIN {X 0,Y 301.844,Z 450.583,A -85,B 0,C 180,E1 -18406.482,E2 -18406.482} C_VEL
LIN {X 0,Y 299.081,Z 466.396,A -85,B 0,C 180,E1 -18407.273,E2 -18407.273} C_VEL
LIN {X 0,Y 295.778,Z 481.845,A -85,B 0,C 180,E1 -18408.295,E2 -18408.295} C_VEL
LIN {X 0,Y 292.206,Z 496.242,A -85,B 0,C 180,E1 -18409.505,E2 -18409.505} C_VEL
LIN {X 0,Y 287.766,Z 511.361,A -85,B 0,C 180,E1 -18411.078,E2 -18411.078} C_VEL
LIN {X 0,Y 283.548,Z 524.45,A -85,B 0,C 180,E1 -18412.781,E2 -18412.781} C_VEL
LIN {X 0,Y 279.318,Z 536.459,A -85,B 0,C 180,E1 -18414.641,E2 -18414.641} C_VEL
LIN {X 0,Y 275.15,Z 547.584,A -85,B 0,C 180,E1 -18416.691,E2 -18416.691} C_VEL
LIN {X 0,Y 270.794,Z 558.7,A -85,B 0,C 180,E1 -18419.165,E2 -18419.165} C_VEL
LIN {X 0,Y 266.425,Z 569.518,A -85,B 0,C 180,E1 -18422.082,E2 -18422.082} C_VEL
LIN {X 0,Y 263.173,Z 577.633,A -85,B 0,C 180,E1 -18424.706,E2 -18424.706} C_VEL
LIN {X 0,Y 260.15,Z 585.422,A -85,B 0,C 180,E1 -18427.778,E2 -18427.778} C_VEL
LIN {X 0,Y 257.763,Z 591.938,A -85,B 0,C 180,E1 -18430.903,E2 -18430.903} C_VEL
LIN {X 0,Y 255.998,Z 597.304,A -85,B 0,C 180,E1 -18434.066,E2 -18434.066} C_VEL
LIN {X 0,Y 254.85,Z 601.49,A -85,B 0,C 180,E1 -18437.255,E2 -18437.255} C_VEL
LIN {X 0,Y 254.179,Z 604.72,A -85,B 0,C 180,E1 -18440.451,E2 -18440.451} C_VEL
LIN {X 0,Y 253.944,Z 606.852,A -85,B 0,C 180,E1 -18443.645,E2 -18443.645} C_VEL
LIN {X 0,Y 253.938,Z 608.093,A -85,B 0,C 180,E1 -18446.827,E2 -18446.827} C_VEL
LIN {X 0,Y 254.054,Z 608.26,A -85,B 0,C 180,E1 -18450,E2 -18450} C_VEL
LIN {X 0,Y 253.966,Z 607.524,A -85,B 0,C 180,E1 -18453.173,E2 -18453.173} C_VEL
LIN {X 0,Y 253.945,Z 605.689,A -85,B 0,C 180,E1 -18456.356,E2 -18456.356} C_VEL
LIN {X 0,Y 254.173,Z 602.909,A -85,B 0,C 180,E1 -18459.55,E2 -18459.55} C_VEL
LIN {X 0,Y 255.057,Z 597.872,A -85,B 0,C 180,E1 -18463.546,E2 -18463.546} C_VEL
LIN {X 0,Y 256.214,Z 592.643,A -85,B 0,C 180,E1 -18466.657,E2 -18466.657} C_VEL
LIN {X 0,Y 258.042,Z 585.914,A -85,B 0,C 180,E1 -18469.904,E2 -18469.904} C_VEL
LIN {X 0,Y 260.429,Z 578.115,A -85,B 0,C 180,E1 -18472.986,E2 -18472.986} C_VEL
LIN {X 0,Y 263.503,Z 568.411,A -85,B 0,C 180,E1 -18476.109,E2 -18476.109} C_VEL
LIN {X 0,Y 266.831,Z 558.5,A -85,B 0,C 180,E1 -18478.73,E2 -18478.73} C_VEL
LIN {X 0,Y 270.472,Z 546.891,A -85,B 0,C 180,E1 -18481.311,E2 -18481.311} C_VEL
LIN {X 0,Y 274.417,Z 534.235,A -85,B 0,C 180,E1 -18483.63,E2 -18483.63} C_VEL
LIN {X 0,Y 278.435,Z 520.649,A -85,B 0,C 180,E1 -18485.677,E2 -18485.677} C_VEL
LIN {X 0,Y 282.492,Z 505.29,A -85,B 0,C 180,E1 -18487.555,E2 -18487.555} C_VEL
LIN {X 0,Y 286.066,Z 490.239,A -85,B 0,C 180,E1 -18489.017,E2 -18489.017} C_VEL
LIN {X 0,Y 289.066,Z 474.848,A -85,B 0,C 180,E1 -18490.226,E2 -18490.226} C_VEL
LIN {X 0,Y 291.708,Z 458.623,A -85,B 0,C 180,E1 -18491.207,E2 -18491.207} C_VEL
LIN {X 0,Y 293.888,Z 442.122,A -85,B 0,C 180,E1 -18491.92,E2 -18491.92} C_VEL
LIN {X 0,Y 295.174,Z 427.115,A -85,B 0,C 180,E1 -18492.373,E2 -18492.373} C_VEL
LIN {X 0,Y 301.716,Z 303.878,A -85,B 0,C 180,E1 -18495.341,E2 -18495.341} C_VEL
LIN {X 0,Y 293.227,Z 286.113,A -85,B 0,C 180,E1 -18497.442,E2 -18497.442} C_VEL
LIN {X 0,Y 284.662,Z 270.287,A -85,B 0,C 180,E1 -18499.668,E2 -18499.668} C_VEL
LIN {X 0,Y 276.854,Z 257.021,A -85,B 0,C 180,E1 -18501.832,E2 -18501.832} C_VEL
LIN {X 0,Y 270.564,Z 246.95,A -85,B 0,C 180,E1 -18503.698,E2 -18503.698} C_VEL
LIN {X 0,Y 265.503,Z 239.471,A -85,B 0,C 180,E1 -18505.272,E2 -18505.272} C_VEL
LIN {X 0,Y 262.909,Z 235.798,A -85,B 0,C 180,E1 -18506.114,E2 -18506.114} C_VEL
LIN {X 0,Y 260.46,Z 232.793,A -85,B 0,C 180,E1 -18506.911,E2 -18506.911} C_VEL
LIN {X 0,Y 259.612,Z 231.16,A -85,B 0,C 180,E1 -18507.22,E2 -18507.22} C_VEL
LIN {X 0,Y 257.39,Z 229.131,A -85,B 0,C 180,E1 -18507.942,E2 -18507.942} C_VEL
LIN {X 0,Y 256.283,Z 226.819,A -85,B 0,C 180,E1 -18508.373,E2 -18508.373} C_VEL
LIN {X 0,Y 256.101,Z 225.87,A -85,B 0,C 180,E1 -18508.506,E2 -18508.506} C_VEL
LIN {X 0,Y 256.14,Z 225.877,A -85,B 0,C 180,E1 -18512.196,E2 -18512.196} C_VEL
LIN {X 0,Y 256.166,Z 225.869,A -85,B 0,C 180,E1 -18515.699,E2 -18515.699} C_VEL
LIN {X 0,Y 256.16,Z 225.863,A -85,B 0,C 180,E1 -18519.104,E2 -18519.104} C_VEL
LIN {X 0,Y 256.244,Z 225.879,A -85,B 0,C 180,E1 -18524.082,E2 -18524.082} C_VEL
LIN {X 0,Y 256.278,Z 225.828,A -85,B 0,C 180,E1 -18528.933,E2 -18528.933} C_VEL
LIN {X 0,Y 256.503,Z 225.846,A -85,B 0,C 180,E1 -18532.126,E2 -18532.126} C_VEL
LIN {X 0,Y 256.492,Z 225.791,A -85,B 0,C 180,E1 -18536.859,E2 -18536.859} C_VEL
LIN {X 0,Y 256.757,Z 225.799,A -85,B 0,C 180,E1 -18540,E2 -18540} C_VEL
LIN {X 0,Y 256.495,Z 225.835,A -85,B 0,C 180,E1 -18543.141,E2 -18543.141} C_VEL
LIN {X 0,Y 256.515,Z 225.842,A -85,B 0,C 180,E1 -18547.874,E2 -18547.874} C_VEL
LIN {X 0,Y 256.293,Z 225.844,A -85,B 0,C 180,E1 -18552.672,E2 -18552.672} C_VEL
LIN {X 0,Y 256.282,Z 225.867,A -85,B 0,C 180,E1 -18556.302,E2 -18556.302} C_VEL
LIN {X 0,Y 256.157,Z 225.883,A -85,B 0,C 180,E1 -18561.12,E2 -18561.12} C_VEL
LIN {X 0,Y 256.189,Z 225.858,A -85,B 0,C 180,E1 -18565.139,E2 -18565.139} C_VEL
LIN {X 0,Y 256.116,Z 225.891,A -85,B 0,C 180,E1 -18569.599,E2 -18569.599} C_VEL
LIN {X 0,Y 256.067,Z 225.882,A -85,B 0,C 180,E1 -18573.293,E2 -18573.293} C_VEL
LIN {X 0,Y 256.113,Z 225.875,A -85,B 0,C 180,E1 -18577.27,E2 -18577.27} C_VEL
LIN {X 0,Y 256.055,Z 225.904,A -85,B 0,C 180,E1 -18581.203,E2 -18581.203} C_VEL
LIN {X 0,Y 256.053,Z 225.896,A -85,B 0,C 180,E1 -18585.531,E2 -18585.531} C_VEL
LIN {X 0,Y 256.053,Z 225.884,A -85,B 0,C 180,E1 -18588.796,E2 -18588.796} C_VEL
LIN {X 0,Y 256.13,Z 225.878,A -85,B 0,C 180,E1 -18592.867,E2 -18592.867} C_VEL
LIN {X 0,Y 256.068,Z 225.901,A -85,B 0,C 180,E1 -18596.707,E2 -18596.707} C_VEL
LIN {X 0,Y 256.112,Z 226.038,A -85,B 0,C 180,E1 -18598.064,E2 -18598.064} C_VEL
LIN {X 0,Y 257.067,Z 228.696,A -85,B 0,C 180,E1 -18598.469,E2 -18598.469} C_VEL
LIN {X 0,Y 259.241,Z 230.938,A -85,B 0,C 180,E1 -18599.189,E2 -18599.189} C_VEL
LIN {X 0,Y 259.934,Z 231.711,A -85,B 0,C 180,E1 -18599.416,E2 -18599.416} C_VEL
